// TIA Portal project "Metrou_2026" (V15.1)

(* hardware
DEVICE "S71500/ET200MP station_1"  S7-1500 station
   slot 0: "Rail_0"  Rack  6ES7 590-1***0-0AA0
   slot 1: "PLC_1(Scari)"  CPU 1513-1 PN  6ES7 513-1AL02-0AB0  V2.6
      slot 3: "CPU display_1"  6ES7591-1AA00-0AA0
DEVICE "S71500/ET200MP station_2"  S7-1500 station
   slot 0: "Rail_0"  Rack  6ES7 590-1***0-0AA0
   slot 1: "PLC_1(Metrou)"  CPU 1513-1 PN  6ES7 513-1AL02-0AB0  V2.6
      slot 3: "CPU display_1"  6ES7591-1AA00-0AA0
DEVICE "HMI_1(Scari)"  KTP900 Basic PN
   slot 0: "HMI_1(Scari)"  KTP900 Basic PN  6AV2 123-2JB03-0AX0  15.1.0.0
   slot 1: "HMI_RT_1"  KTP900 Basic PN  6AV2 123-2JB03-0AX0  15.1.0.0
   slot 5: "HMI_1(Scari).IE_CP_1"  PROFINET Interface  15.0.1.0
      slot 1: "PROFINET Interface_1"  PROFINET Interface
         slot 1: "Port_1"  Port
DEVICE "HMI_1(Metrou)"  KTP900 Basic PN
   slot 0: "HMI_1(Metrou)"  KTP900 Basic PN  6AV2 123-2JB03-0AX0  15.1.0.0
   slot 1: "HMI_RT_2"  KTP900 Basic PN  6AV2 123-2JB03-0AX0  15.1.0.0
   slot 5: "HMI_1(Metrou).IE_CP_1"  PROFINET Interface  15.0.1.0
      slot 1: "PROFINET Interface_1"  PROFINET Interface
         slot 1: "Port_1"  Port
*)

// ===== PLC "PLC_1(Scari)"  CPU 1513-1 PN =====

// folder: Alarme/Avarii

DATA_BLOCK "Alarme"   // DB1
{ S7_Optimized_Access := 'TRUE' }
VERSION : 0.1
   VAR
      gather : Word;
      "array" : Array[0..15] of Bool;
   END_VAR
BEGIN
END_DATA_BLOCK

DATA_BLOCK "Avarii"   // DB2
{ S7_Optimized_Access := 'TRUE' }
VERSION : 0.1
   VAR
      esd : Bool;
      btn_esd : Bool;
      reset_esd : Bool;
      avarie_1 : Bool;
      avarie_2 : Bool;
      avarie_3 : Bool;
      avarie_4 : Bool;
      btn_avarie_1 : Bool;
      btn_avarie_2 : Bool;
      btn_avarie_3 : Bool;
      btn_avarie_4 : Bool;
      reset_avarie_1 : Bool;
      reset_avarie_2 : Bool;
      reset_avarie_3 : Bool;
      reset_avarie_4 : Bool;
   END_VAR
BEGIN
END_DATA_BLOCK

// folder: HMI

DATA_BLOCK "HMI"   // DB10
{ S7_Optimized_Access := 'TRUE' }
VERSION : 0.1
   VAR
      motor_stea_1 : Bool;
      motor_triunghi_1 : Bool;
      mod_motor_1 : DInt;   // 0 -> stea, 1 -> triunghi
      pornit_HMI_1 : Bool;
      time_elapsed_HMI_1 : Bool;
      timp_secunde_c_1 : Time;
      timp_secunde_u_1 : Time;
      motor_stea_2 : Bool;
      motor_triunghi_2 : Bool;
      mod_motor_2 : DInt;   // 0 -> stea, 1 -> triunghi
      pornit_HMI_2 : Bool;
      time_elapsed_HMI_2 : Bool;
      timp_secunde_c_2 : Time;
      timp_secunde_u_2 : Time;
      motor_stea_3 : Bool;
      motor_triunghi_3 : Bool;
      mod_motor_3 : DInt;   // 0 -> stea, 1 -> triunghi
      pornit_HMI_3 : Bool;
      time_elapsed_HMI_3 : Bool;
      timp_secunde_c_3 : Time;
      timp_secunde_u_3 : Time;
      motor_stea_4 : Bool;
      motor_triunghi_4 : Bool;
      mod_motor_4 : DInt;   // 0 -> stea, 1 -> triunghi
      pornit_HMI_4 : Bool;
      time_elapsed_HMI_4 : Bool;
      timp_secunde_c_4 : Time;
      timp_secunde_u_4 : Time;
   END_VAR
BEGIN
END_DATA_BLOCK

// folder: Instante

DATA_BLOCK "ESD_Instanta"   // DB4
{ S7_Optimized_Access := 'TRUE' }
VERSION : 0.1
// stored: InstanceOfName Avarei/ESD_FB
"Avarei/ESD_FB"
BEGIN
END_DATA_BLOCK

DATA_BLOCK "Scara1_Instanta_Alarme"   // DB5
{ S7_Optimized_Access := 'TRUE' }
VERSION : 0.1
// stored: InstanceOfName Avarei/ESD_FB
"Avarei/ESD_FB"
BEGIN
END_DATA_BLOCK

DATA_BLOCK "Scara2_Instanta_Alarme"   // DB6
{ S7_Optimized_Access := 'TRUE' }
VERSION : 0.1
// stored: InstanceOfName Avarei/ESD_FB
"Avarei/ESD_FB"
BEGIN
END_DATA_BLOCK

DATA_BLOCK "Scara3_Instanta_Alarme"   // DB7
{ S7_Optimized_Access := 'TRUE' }
VERSION : 0.1
// stored: InstanceOfName Avarei/ESD_FB
"Avarei/ESD_FB"
BEGIN
END_DATA_BLOCK

DATA_BLOCK "Scara4_Instanta_Alarme"   // DB8
{ S7_Optimized_Access := 'TRUE' }
VERSION : 0.1
// stored: InstanceOfName Avarei/ESD_FB
"Avarei/ESD_FB"
BEGIN
END_DATA_BLOCK

DATA_BLOCK "Scara1_Instanta_FB"   // DB9
{ S7_Optimized_Access := 'TRUE' }
VERSION : 0.1
// stored: InstanceOfName Scari
"Scari"
BEGIN
END_DATA_BLOCK

DATA_BLOCK "HMI_Scara_Instanta"   // DB11
{ S7_Optimized_Access := 'TRUE' }
VERSION : 0.1
// stored: InstanceOfName HMI_Scara
"HMI_Scara"
BEGIN
END_DATA_BLOCK

DATA_BLOCK "Scara2_Instanta_FB"   // DB15
{ S7_Optimized_Access := 'TRUE' }
VERSION : 0.1
// stored: InstanceOfName Scari
"Scari"
BEGIN
END_DATA_BLOCK

DATA_BLOCK "Scara4_Instanta_FB"   // DB16
{ S7_Optimized_Access := 'TRUE' }
VERSION : 0.1
// stored: InstanceOfName Scari
"Scari"
BEGIN
END_DATA_BLOCK

DATA_BLOCK "Scara3_Instanta_FB"   // DB17
{ S7_Optimized_Access := 'TRUE' }
VERSION : 0.1
// stored: InstanceOfName Scari
"Scari"
BEGIN
END_DATA_BLOCK

DATA_BLOCK "HMI_Scara2_Instanta"   // DB18
{ S7_Optimized_Access := 'TRUE' }
VERSION : 0.1
// stored: InstanceOfName HMI_Scara
"HMI_Scara"
BEGIN
END_DATA_BLOCK

DATA_BLOCK "HMI_Scara3_Instanta"   // DB19
{ S7_Optimized_Access := 'TRUE' }
VERSION : 0.1
// stored: InstanceOfName HMI_Scara
"HMI_Scara"
BEGIN
END_DATA_BLOCK

DATA_BLOCK "HMI_Scara4_Instanta"   // DB20
{ S7_Optimized_Access := 'TRUE' }
VERSION : 0.1
// stored: InstanceOfName HMI_Scara
"HMI_Scara"
BEGIN
END_DATA_BLOCK

// folder: Scari

DATA_BLOCK "Scara1_DB"   // DB3
{ S7_Optimized_Access := 'TRUE' }
VERSION : 0.1
   VAR
      "mod" : DInt;
      btn_start : Bool;
      btn_stop : Bool;
      senzor_persoana_urcare : Bool;
      senzor_persoana_coborare : Bool;
      stea_urcare : Bool;
      stea_coborare : Bool;
      triunghi_urcare : Bool;
      triunghi_coborare : Bool;
      urcare_HMI : Bool;
      coborare_HMI : Bool;
      et_stea_u : Time;
      et_stea_c : Time;
      et_persoana_u : Time;
      et_persoana_c : Time;
   END_VAR
BEGIN
END_DATA_BLOCK

DATA_BLOCK "Scara2_DB"   // DB12
{ S7_Optimized_Access := 'TRUE' }
VERSION : 0.1
   VAR
      "mod" : DInt;
      btn_start : Bool;
      btn_stop : Bool;
      senzor_persoana_urcare : Bool;
      senzor_persoana_coborare : Bool;
      stea_urcare : Bool;
      stea_coborare : Bool;
      triunghi_urcare : Bool;
      triunghi_coborare : Bool;
      urcare_HMI : Bool;
      coborare_HMI : Bool;
      et_stea_u : Time;
      et_stea_c : Time;
      et_persoana_u : Time;
      et_persoana_c : Time;
   END_VAR
BEGIN
END_DATA_BLOCK

DATA_BLOCK "Scara3_DB"   // DB13
{ S7_Optimized_Access := 'TRUE' }
VERSION : 0.1
   VAR
      "mod" : DInt;
      btn_start : Bool;
      btn_stop : Bool;
      senzor_persoana_urcare : Bool;
      senzor_persoana_coborare : Bool;
      stea_urcare : Bool;
      stea_coborare : Bool;
      triunghi_urcare : Bool;
      triunghi_coborare : Bool;
      urcare_HMI : Bool;
      coborare_HMI : Bool;
      et_stea_u : Time;
      et_stea_c : Time;
      et_persoana_u : Time;
      et_persoana_c : Time;
   END_VAR
BEGIN
END_DATA_BLOCK

DATA_BLOCK "Scara4_DB"   // DB14
{ S7_Optimized_Access := 'TRUE' }
VERSION : 0.1
   VAR
      "mod" : DInt;
      btn_start : Bool;
      btn_stop : Bool;
      senzor_persoana_urcare : Bool;
      senzor_persoana_coborare : Bool;
      stea_urcare : Bool;
      stea_coborare : Bool;
      triunghi_urcare : Bool;
      triunghi_coborare : Bool;
      urcare_HMI : Bool;
      coborare_HMI : Bool;
      et_stea_u : Time;
      et_stea_c : Time;
      et_persoana_u : Time;
      et_persoana_c : Time;
   END_VAR
BEGIN
END_DATA_BLOCK

// folder: (top level)

ORGANIZATION_BLOCK "Main"   // OB1, LAD, ProgramCycle
TITLE = "Main Program Sweep (Cycle)"
{ S7_Optimized_Access := 'TRUE' }
VERSION : 0.1
   VAR_INPUT
      Initial_Call : Bool;   // Initial call of this OB
      Remanence : Bool;   // =True, if remanent data are available
   END_VAR
BEGIN

REGION Network 1: gather de alarme
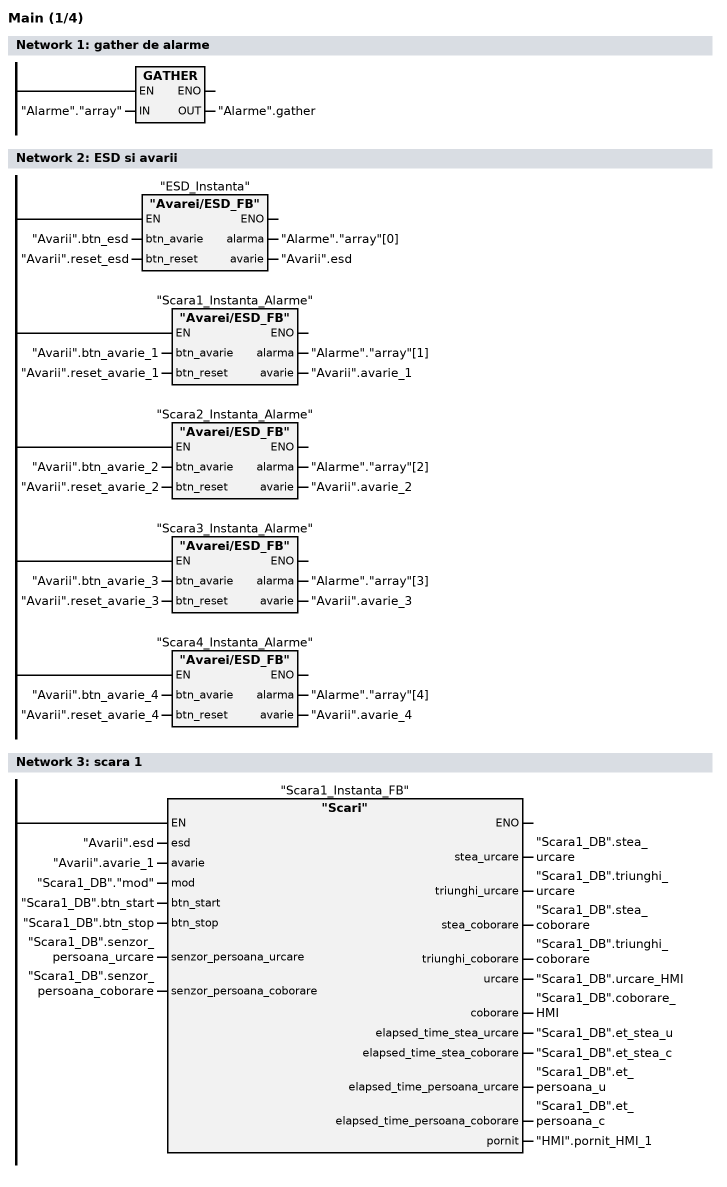
   GATHER(IN := "Alarme"."array", OUT => "Alarme".gather);
END_REGION

REGION Network 2: ESD si avarii
   RUNG wire#powerrail
      "ESD_Instanta"(btn_avarie := "Avarii".btn_esd, btn_reset := "Avarii".reset_esd, alarma => "Alarme"."array"[0], avarie => "Avarii".esd)
   END_RUNG
   RUNG wire#powerrail
      "Scara1_Instanta_Alarme"(btn_avarie := "Avarii".btn_avarie_1, btn_reset := "Avarii".reset_avarie_1, alarma => "Alarme"."array"[1], avarie => "Avarii".avarie_1)
   END_RUNG
   RUNG wire#powerrail
      "Scara2_Instanta_Alarme"(btn_avarie := "Avarii".btn_avarie_2, btn_reset := "Avarii".reset_avarie_2, alarma => "Alarme"."array"[2], avarie => "Avarii".avarie_2)
   END_RUNG
   RUNG wire#powerrail
      "Scara3_Instanta_Alarme"(btn_avarie := "Avarii".btn_avarie_3, btn_reset := "Avarii".reset_avarie_3, alarma => "Alarme"."array"[3], avarie => "Avarii".avarie_3)
   END_RUNG
   RUNG wire#powerrail
      "Scara4_Instanta_Alarme"(btn_avarie := "Avarii".btn_avarie_4, btn_reset := "Avarii".reset_avarie_4, alarma => "Alarme"."array"[4], avarie => "Avarii".avarie_4)
   END_RUNG
   // the same network as SCL:
   "ESD_Instanta"(btn_avarie := "Avarii".btn_esd,   // "Avarei/ESD_FB"
                  btn_reset := "Avarii".reset_esd,
                  alarma => "Alarme"."array"[0],
                  avarie => "Avarii".esd);
   "Scara1_Instanta_Alarme"(btn_avarie := "Avarii".btn_avarie_1,   // "Avarei/ESD_FB"
                           btn_reset := "Avarii".reset_avarie_1,
                           alarma => "Alarme"."array"[1],
                           avarie => "Avarii".avarie_1);
   "Scara2_Instanta_Alarme"(btn_avarie := "Avarii".btn_avarie_2,   // "Avarei/ESD_FB"
                           btn_reset := "Avarii".reset_avarie_2,
                           alarma => "Alarme"."array"[2],
                           avarie => "Avarii".avarie_2);
   "Scara3_Instanta_Alarme"(btn_avarie := "Avarii".btn_avarie_3,   // "Avarei/ESD_FB"
                           btn_reset := "Avarii".reset_avarie_3,
                           alarma => "Alarme"."array"[3],
                           avarie => "Avarii".avarie_3);
   "Scara4_Instanta_Alarme"(btn_avarie := "Avarii".btn_avarie_4,   // "Avarei/ESD_FB"
                           btn_reset := "Avarii".reset_avarie_4,
                           alarma => "Alarme"."array"[4],
                           avarie => "Avarii".avarie_4);
END_REGION

REGION Network 3: scara 1
   RUNG wire#powerrail
      "Scara1_Instanta_FB"(esd := "Avarii".esd, avarie := "Avarii".avarie_1, "mod" := "Scara1_DB"."mod", btn_start := "Scara1_DB".btn_start, btn_stop := "Scara1_DB".btn_stop, senzor_persoana_urcare := "Scara1_DB".senzor_persoana_urcare, senzor_persoana_coborare := "Scara1_DB".senzor_persoana_coborare, stea_urcare => "Scara1_DB".stea_urcare, triunghi_urcare => "Scara1_DB".triunghi_urcare, stea_coborare => "Scara1_DB".stea_coborare, triunghi_coborare => "Scara1_DB".triunghi_coborare, urcare => "Scara1_DB".urcare_HMI, coborare => "Scara1_DB".coborare_HMI, elapsed_time_stea_urcare => "Scara1_DB".et_stea_u, elapsed_time_stea_coborare => "Scara1_DB".et_stea_c, elapsed_time_persoana_urcare => "Scara1_DB".et_persoana_u, elapsed_time_persoana_coborare => "Scara1_DB".et_persoana_c, pornit => "HMI".pornit_HMI_1)
   END_RUNG
   // the same network as SCL:
   "Scara1_Instanta_FB"(esd := "Avarii".esd,   // "Scari"
                        avarie := "Avarii".avarie_1,
                        "mod" := "Scara1_DB"."mod",
                        btn_start := "Scara1_DB".btn_start,
                        btn_stop := "Scara1_DB".btn_stop,
                        senzor_persoana_urcare := "Scara1_DB".senzor_persoana_urcare,
                        senzor_persoana_coborare := "Scara1_DB".senzor_persoana_coborare,
                        stea_urcare => "Scara1_DB".stea_urcare,
                        triunghi_urcare => "Scara1_DB".triunghi_urcare,
                        stea_coborare => "Scara1_DB".stea_coborare,
                        triunghi_coborare => "Scara1_DB".triunghi_coborare,
                        urcare => "Scara1_DB".urcare_HMI,
                        coborare => "Scara1_DB".coborare_HMI,
                        elapsed_time_stea_urcare => "Scara1_DB".et_stea_u,
                        elapsed_time_stea_coborare => "Scara1_DB".et_stea_c,
                        elapsed_time_persoana_urcare => "Scara1_DB".et_persoana_u,
                        elapsed_time_persoana_coborare => "Scara1_DB".et_persoana_c,
                        pornit => "HMI".pornit_HMI_1);
END_REGION

REGION Network 4: HMI scara 1
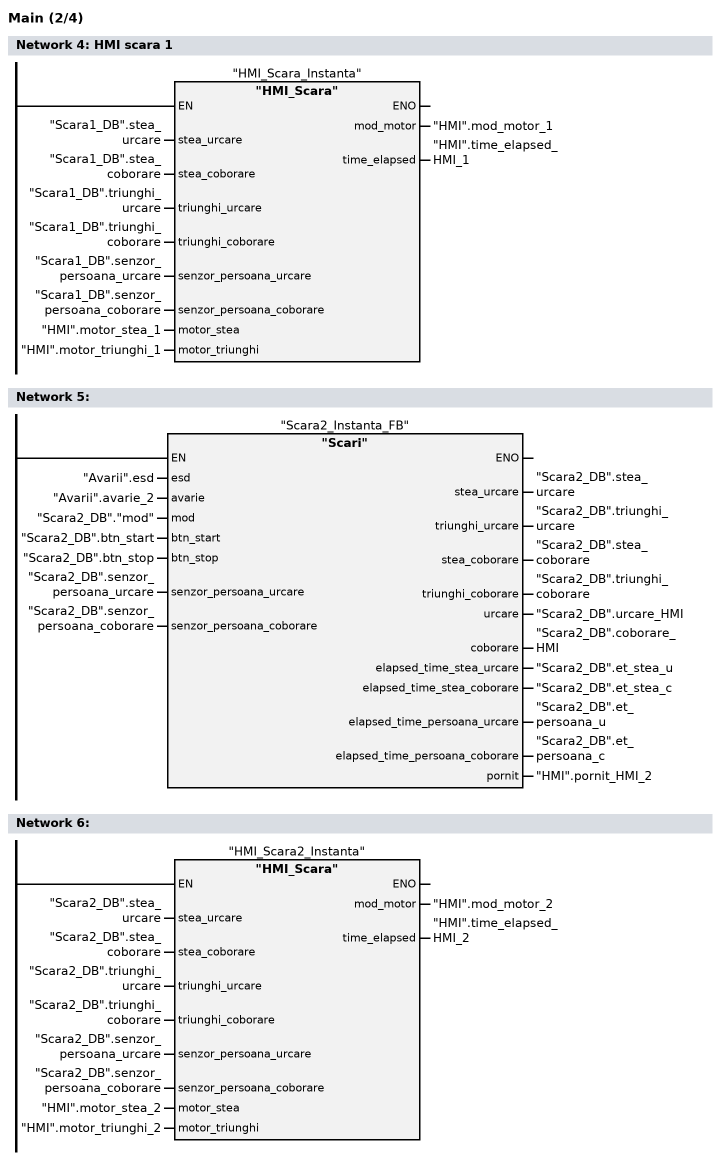
   RUNG wire#powerrail
      "HMI_Scara_Instanta"(stea_urcare := "Scara1_DB".stea_urcare, stea_coborare := "Scara1_DB".stea_coborare, triunghi_urcare := "Scara1_DB".triunghi_urcare, triunghi_coborare := "Scara1_DB".triunghi_coborare, senzor_persoana_urcare := "Scara1_DB".senzor_persoana_urcare, senzor_persoana_coborare := "Scara1_DB".senzor_persoana_coborare, motor_stea := "HMI".motor_stea_1, motor_triunghi := "HMI".motor_triunghi_1, mod_motor => "HMI".mod_motor_1, time_elapsed => "HMI".time_elapsed_HMI_1)
   END_RUNG
   // the same network as SCL:
   "HMI_Scara_Instanta"(stea_urcare := "Scara1_DB".stea_urcare,   // "HMI_Scara"
                        stea_coborare := "Scara1_DB".stea_coborare,
                        triunghi_urcare := "Scara1_DB".triunghi_urcare,
                        triunghi_coborare := "Scara1_DB".triunghi_coborare,
                        senzor_persoana_urcare := "Scara1_DB".senzor_persoana_urcare,
                        senzor_persoana_coborare := "Scara1_DB".senzor_persoana_coborare,
                        motor_stea := "HMI".motor_stea_1,
                        motor_triunghi := "HMI".motor_triunghi_1,
                        mod_motor => "HMI".mod_motor_1,
                        time_elapsed => "HMI".time_elapsed_HMI_1);
END_REGION

REGION Network 5
   RUNG wire#powerrail
      "Scara2_Instanta_FB"(esd := "Avarii".esd, avarie := "Avarii".avarie_2, "mod" := "Scara2_DB"."mod", btn_start := "Scara2_DB".btn_start, btn_stop := "Scara2_DB".btn_stop, senzor_persoana_urcare := "Scara2_DB".senzor_persoana_urcare, senzor_persoana_coborare := "Scara2_DB".senzor_persoana_coborare, stea_urcare => "Scara2_DB".stea_urcare, triunghi_urcare => "Scara2_DB".triunghi_urcare, stea_coborare => "Scara2_DB".stea_coborare, triunghi_coborare => "Scara2_DB".triunghi_coborare, urcare => "Scara2_DB".urcare_HMI, coborare => "Scara2_DB".coborare_HMI, elapsed_time_stea_urcare => "Scara2_DB".et_stea_u, elapsed_time_stea_coborare => "Scara2_DB".et_stea_c, elapsed_time_persoana_urcare => "Scara2_DB".et_persoana_u, elapsed_time_persoana_coborare => "Scara2_DB".et_persoana_c, pornit => "HMI".pornit_HMI_2)
   END_RUNG
   // the same network as SCL:
   "Scara2_Instanta_FB"(esd := "Avarii".esd,   // "Scari"
                        avarie := "Avarii".avarie_2,
                        "mod" := "Scara2_DB"."mod",
                        btn_start := "Scara2_DB".btn_start,
                        btn_stop := "Scara2_DB".btn_stop,
                        senzor_persoana_urcare := "Scara2_DB".senzor_persoana_urcare,
                        senzor_persoana_coborare := "Scara2_DB".senzor_persoana_coborare,
                        stea_urcare => "Scara2_DB".stea_urcare,
                        triunghi_urcare => "Scara2_DB".triunghi_urcare,
                        stea_coborare => "Scara2_DB".stea_coborare,
                        triunghi_coborare => "Scara2_DB".triunghi_coborare,
                        urcare => "Scara2_DB".urcare_HMI,
                        coborare => "Scara2_DB".coborare_HMI,
                        elapsed_time_stea_urcare => "Scara2_DB".et_stea_u,
                        elapsed_time_stea_coborare => "Scara2_DB".et_stea_c,
                        elapsed_time_persoana_urcare => "Scara2_DB".et_persoana_u,
                        elapsed_time_persoana_coborare => "Scara2_DB".et_persoana_c,
                        pornit => "HMI".pornit_HMI_2);
END_REGION

REGION Network 6
   RUNG wire#powerrail
      "HMI_Scara2_Instanta"(stea_urcare := "Scara2_DB".stea_urcare, stea_coborare := "Scara2_DB".stea_coborare, triunghi_urcare := "Scara2_DB".triunghi_urcare, triunghi_coborare := "Scara2_DB".triunghi_coborare, senzor_persoana_urcare := "Scara2_DB".senzor_persoana_urcare, senzor_persoana_coborare := "Scara2_DB".senzor_persoana_coborare, motor_stea := "HMI".motor_stea_2, motor_triunghi := "HMI".motor_triunghi_2, mod_motor => "HMI".mod_motor_2, time_elapsed => "HMI".time_elapsed_HMI_2)
   END_RUNG
   // the same network as SCL:
   "HMI_Scara2_Instanta"(stea_urcare := "Scara2_DB".stea_urcare,   // "HMI_Scara"
                         stea_coborare := "Scara2_DB".stea_coborare,
                         triunghi_urcare := "Scara2_DB".triunghi_urcare,
                         triunghi_coborare := "Scara2_DB".triunghi_coborare,
                         senzor_persoana_urcare := "Scara2_DB".senzor_persoana_urcare,
                         senzor_persoana_coborare := "Scara2_DB".senzor_persoana_coborare,
                         motor_stea := "HMI".motor_stea_2,
                         motor_triunghi := "HMI".motor_triunghi_2,
                         mod_motor => "HMI".mod_motor_2,
                         time_elapsed => "HMI".time_elapsed_HMI_2);
END_REGION

REGION Network 7
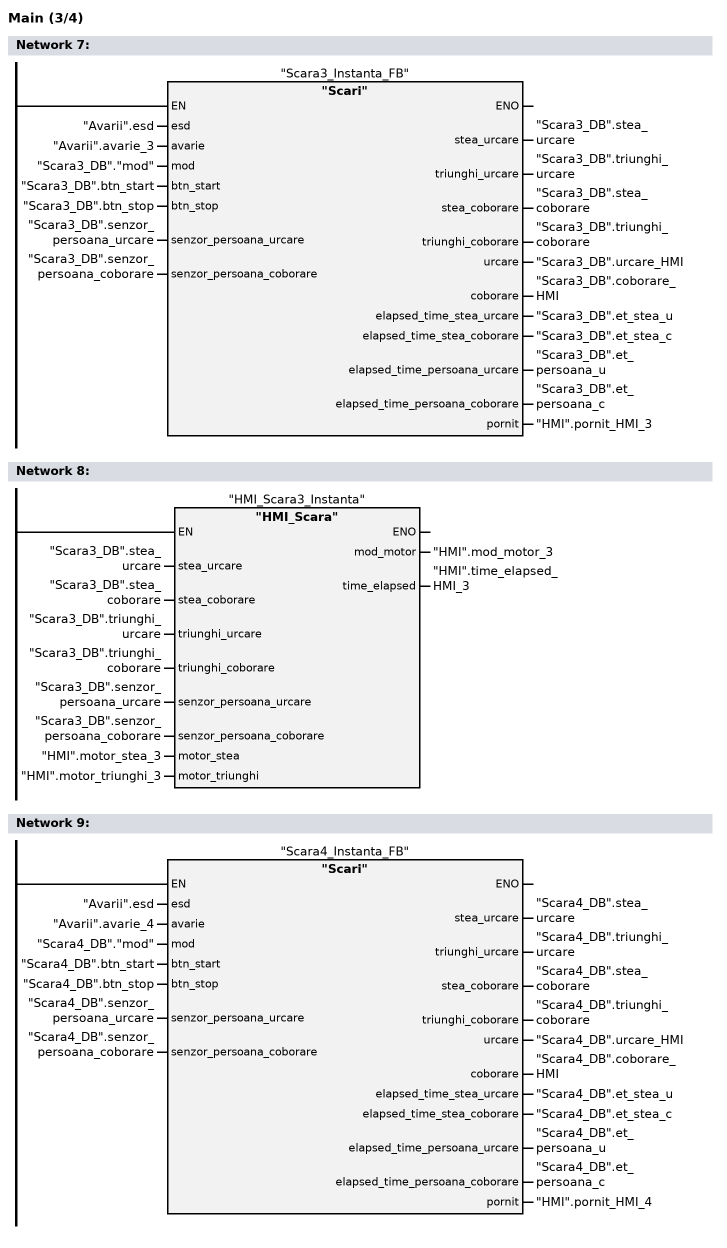
   RUNG wire#powerrail
      "Scara3_Instanta_FB"(esd := "Avarii".esd, avarie := "Avarii".avarie_3, "mod" := "Scara3_DB"."mod", btn_start := "Scara3_DB".btn_start, btn_stop := "Scara3_DB".btn_stop, senzor_persoana_urcare := "Scara3_DB".senzor_persoana_urcare, senzor_persoana_coborare := "Scara3_DB".senzor_persoana_coborare, stea_urcare => "Scara3_DB".stea_urcare, triunghi_urcare => "Scara3_DB".triunghi_urcare, stea_coborare => "Scara3_DB".stea_coborare, triunghi_coborare => "Scara3_DB".triunghi_coborare, urcare => "Scara3_DB".urcare_HMI, coborare => "Scara3_DB".coborare_HMI, elapsed_time_stea_urcare => "Scara3_DB".et_stea_u, elapsed_time_stea_coborare => "Scara3_DB".et_stea_c, elapsed_time_persoana_urcare => "Scara3_DB".et_persoana_u, elapsed_time_persoana_coborare => "Scara3_DB".et_persoana_c, pornit => "HMI".pornit_HMI_3)
   END_RUNG
   // the same network as SCL:
   "Scara3_Instanta_FB"(esd := "Avarii".esd,   // "Scari"
                        avarie := "Avarii".avarie_3,
                        "mod" := "Scara3_DB"."mod",
                        btn_start := "Scara3_DB".btn_start,
                        btn_stop := "Scara3_DB".btn_stop,
                        senzor_persoana_urcare := "Scara3_DB".senzor_persoana_urcare,
                        senzor_persoana_coborare := "Scara3_DB".senzor_persoana_coborare,
                        stea_urcare => "Scara3_DB".stea_urcare,
                        triunghi_urcare => "Scara3_DB".triunghi_urcare,
                        stea_coborare => "Scara3_DB".stea_coborare,
                        triunghi_coborare => "Scara3_DB".triunghi_coborare,
                        urcare => "Scara3_DB".urcare_HMI,
                        coborare => "Scara3_DB".coborare_HMI,
                        elapsed_time_stea_urcare => "Scara3_DB".et_stea_u,
                        elapsed_time_stea_coborare => "Scara3_DB".et_stea_c,
                        elapsed_time_persoana_urcare => "Scara3_DB".et_persoana_u,
                        elapsed_time_persoana_coborare => "Scara3_DB".et_persoana_c,
                        pornit => "HMI".pornit_HMI_3);
END_REGION

REGION Network 8
   RUNG wire#powerrail
      "HMI_Scara3_Instanta"(stea_urcare := "Scara3_DB".stea_urcare, stea_coborare := "Scara3_DB".stea_coborare, triunghi_urcare := "Scara3_DB".triunghi_urcare, triunghi_coborare := "Scara3_DB".triunghi_coborare, senzor_persoana_urcare := "Scara3_DB".senzor_persoana_urcare, senzor_persoana_coborare := "Scara3_DB".senzor_persoana_coborare, motor_stea := "HMI".motor_stea_3, motor_triunghi := "HMI".motor_triunghi_3, mod_motor => "HMI".mod_motor_3, time_elapsed => "HMI".time_elapsed_HMI_3)
   END_RUNG
   // the same network as SCL:
   "HMI_Scara3_Instanta"(stea_urcare := "Scara3_DB".stea_urcare,   // "HMI_Scara"
                         stea_coborare := "Scara3_DB".stea_coborare,
                         triunghi_urcare := "Scara3_DB".triunghi_urcare,
                         triunghi_coborare := "Scara3_DB".triunghi_coborare,
                         senzor_persoana_urcare := "Scara3_DB".senzor_persoana_urcare,
                         senzor_persoana_coborare := "Scara3_DB".senzor_persoana_coborare,
                         motor_stea := "HMI".motor_stea_3,
                         motor_triunghi := "HMI".motor_triunghi_3,
                         mod_motor => "HMI".mod_motor_3,
                         time_elapsed => "HMI".time_elapsed_HMI_3);
END_REGION

REGION Network 9
   RUNG wire#powerrail
      "Scara4_Instanta_FB"(esd := "Avarii".esd, avarie := "Avarii".avarie_4, "mod" := "Scara4_DB"."mod", btn_start := "Scara4_DB".btn_start, btn_stop := "Scara4_DB".btn_stop, senzor_persoana_urcare := "Scara4_DB".senzor_persoana_urcare, senzor_persoana_coborare := "Scara4_DB".senzor_persoana_coborare, stea_urcare => "Scara4_DB".stea_urcare, triunghi_urcare => "Scara4_DB".triunghi_urcare, stea_coborare => "Scara4_DB".stea_coborare, triunghi_coborare => "Scara4_DB".triunghi_coborare, urcare => "Scara4_DB".urcare_HMI, coborare => "Scara4_DB".coborare_HMI, elapsed_time_stea_urcare => "Scara4_DB".et_stea_u, elapsed_time_stea_coborare => "Scara4_DB".et_stea_c, elapsed_time_persoana_urcare => "Scara4_DB".et_persoana_u, elapsed_time_persoana_coborare => "Scara4_DB".et_persoana_c, pornit => "HMI".pornit_HMI_4)
   END_RUNG
   // the same network as SCL:
   "Scara4_Instanta_FB"(esd := "Avarii".esd,   // "Scari"
                        avarie := "Avarii".avarie_4,
                        "mod" := "Scara4_DB"."mod",
                        btn_start := "Scara4_DB".btn_start,
                        btn_stop := "Scara4_DB".btn_stop,
                        senzor_persoana_urcare := "Scara4_DB".senzor_persoana_urcare,
                        senzor_persoana_coborare := "Scara4_DB".senzor_persoana_coborare,
                        stea_urcare => "Scara4_DB".stea_urcare,
                        triunghi_urcare => "Scara4_DB".triunghi_urcare,
                        stea_coborare => "Scara4_DB".stea_coborare,
                        triunghi_coborare => "Scara4_DB".triunghi_coborare,
                        urcare => "Scara4_DB".urcare_HMI,
                        coborare => "Scara4_DB".coborare_HMI,
                        elapsed_time_stea_urcare => "Scara4_DB".et_stea_u,
                        elapsed_time_stea_coborare => "Scara4_DB".et_stea_c,
                        elapsed_time_persoana_urcare => "Scara4_DB".et_persoana_u,
                        elapsed_time_persoana_coborare => "Scara4_DB".et_persoana_c,
                        pornit => "HMI".pornit_HMI_4);
END_REGION

REGION Network 10
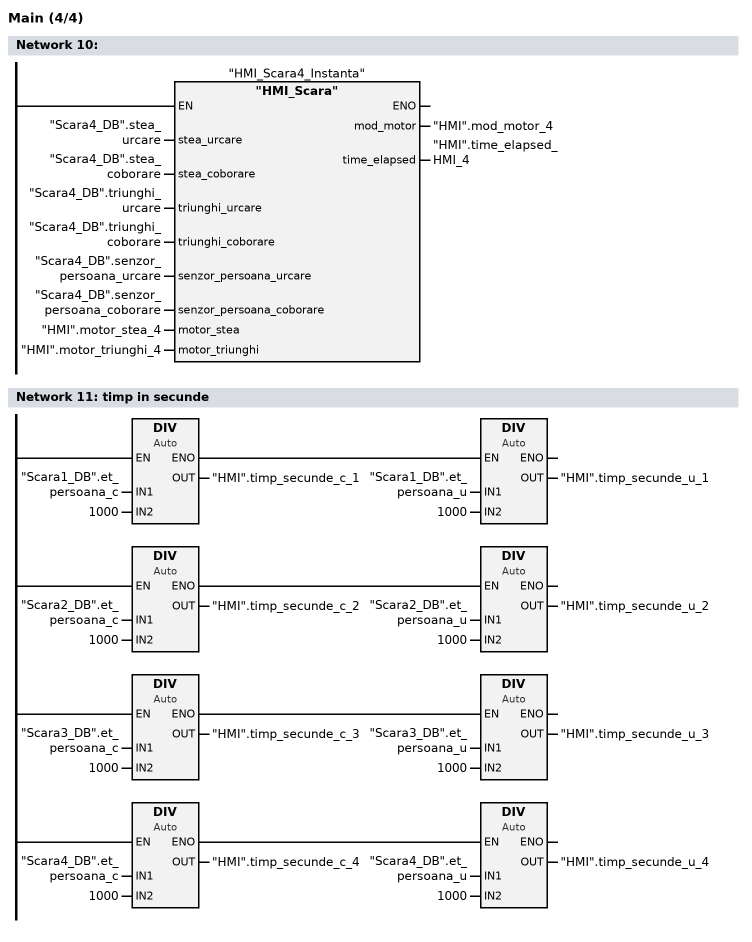
   RUNG wire#powerrail
      "HMI_Scara4_Instanta"(stea_urcare := "Scara4_DB".stea_urcare, stea_coborare := "Scara4_DB".stea_coborare, triunghi_urcare := "Scara4_DB".triunghi_urcare, triunghi_coborare := "Scara4_DB".triunghi_coborare, senzor_persoana_urcare := "Scara4_DB".senzor_persoana_urcare, senzor_persoana_coborare := "Scara4_DB".senzor_persoana_coborare, motor_stea := "HMI".motor_stea_4, motor_triunghi := "HMI".motor_triunghi_4, mod_motor => "HMI".mod_motor_4, time_elapsed => "HMI".time_elapsed_HMI_4)
   END_RUNG
   // the same network as SCL:
   "HMI_Scara4_Instanta"(stea_urcare := "Scara4_DB".stea_urcare,   // "HMI_Scara"
                         stea_coborare := "Scara4_DB".stea_coborare,
                         triunghi_urcare := "Scara4_DB".triunghi_urcare,
                         triunghi_coborare := "Scara4_DB".triunghi_coborare,
                         senzor_persoana_urcare := "Scara4_DB".senzor_persoana_urcare,
                         senzor_persoana_coborare := "Scara4_DB".senzor_persoana_coborare,
                         motor_stea := "HMI".motor_stea_4,
                         motor_triunghi := "HMI".motor_triunghi_4,
                         mod_motor => "HMI".mod_motor_4,
                         time_elapsed => "HMI".time_elapsed_HMI_4);
END_REGION

REGION Network 11: timp in secunde
   RUNG wire#powerrail
      Div(in1 := "Scara1_DB".et_persoana_c, in2 := 1000, out => "HMI".timp_secunde_c_1)
      Div(in1 := "Scara1_DB".et_persoana_u, in2 := 1000, out => "HMI".timp_secunde_u_1)
   END_RUNG
   RUNG wire#powerrail
      Div(in1 := "Scara2_DB".et_persoana_c, in2 := 1000, out => "HMI".timp_secunde_c_2)
      Div(in1 := "Scara2_DB".et_persoana_u, in2 := 1000, out => "HMI".timp_secunde_u_2)
   END_RUNG
   RUNG wire#powerrail
      Div(in1 := "Scara3_DB".et_persoana_c, in2 := 1000, out => "HMI".timp_secunde_c_3)
      Div(in1 := "Scara3_DB".et_persoana_u, in2 := 1000, out => "HMI".timp_secunde_u_3)
   END_RUNG
   RUNG wire#powerrail
      Div(in1 := "Scara4_DB".et_persoana_c, in2 := 1000, out => "HMI".timp_secunde_c_4)
      Div(in1 := "Scara4_DB".et_persoana_u, in2 := 1000, out => "HMI".timp_secunde_u_4)
   END_RUNG
   // the same network as SCL:
   "HMI".timp_secunde_c_1 := "Scara1_DB".et_persoana_c / 1000;
   "HMI".timp_secunde_u_1 := "Scara1_DB".et_persoana_u / 1000;
   "HMI".timp_secunde_c_2 := "Scara2_DB".et_persoana_c / 1000;
   "HMI".timp_secunde_u_2 := "Scara2_DB".et_persoana_u / 1000;
   "HMI".timp_secunde_c_3 := "Scara3_DB".et_persoana_c / 1000;
   "HMI".timp_secunde_u_3 := "Scara3_DB".et_persoana_u / 1000;
   "HMI".timp_secunde_c_4 := "Scara4_DB".et_persoana_c / 1000;
   "HMI".timp_secunde_u_4 := "Scara4_DB".et_persoana_u / 1000;
END_REGION
END_ORGANIZATION_BLOCK

// folder: Alarme/Avarii

FUNCTION_BLOCK "Avarei/ESD_FB"   // FB2, LAD
{ S7_Optimized_Access := 'TRUE' }
VERSION : 0.1
   VAR_OUTPUT
      alarma : Bool;
      avarie : Bool;
   END_VAR
   VAR_IN_OUT
      btn_avarie : Bool;
      btn_reset : Bool;
   END_VAR
   VAR
      ton : TON_TIME;
   END_VAR
BEGIN

REGION Network 1: seteaza avaria
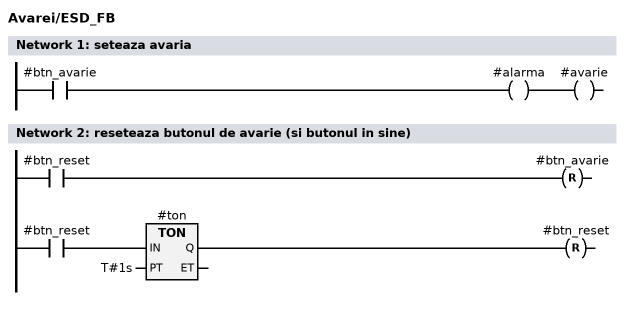
   RUNG wire#powerrail
      Contact( #btn_avarie )
      Coil( #alarma )
      Coil( #avarie )
   END_RUNG
   // the same network as SCL:
   #alarma := #btn_avarie;
   #avarie := #btn_avarie;
END_REGION

REGION Network 2: reseteaza butonul de avarie (si butonul in sine)
   IF #btn_reset THEN #btn_avarie := FALSE; END_IF;
   #ton(IN := #btn_reset, PT := T#1s);   // TON
   IF #ton.Q THEN #btn_reset := FALSE; END_IF;
END_REGION
END_FUNCTION_BLOCK

// folder: HMI

FUNCTION_BLOCK "HMI_Scara"   // FB3, LAD
{ S7_Optimized_Access := 'TRUE' }
VERSION : 0.1
   VAR_INPUT
      stea_urcare : Bool;
      stea_coborare : Bool;
      triunghi_urcare : Bool;
      triunghi_coborare : Bool;
      senzor_persoana_urcare : Bool;
      senzor_persoana_coborare : Bool;
   END_VAR
   VAR_OUTPUT
      mod_motor : DInt;
      time_elapsed : Bool;
   END_VAR
   VAR_IN_OUT
      motor_stea : Bool;
      motor_triunghi : Bool;
   END_VAR
BEGIN

REGION Network 1
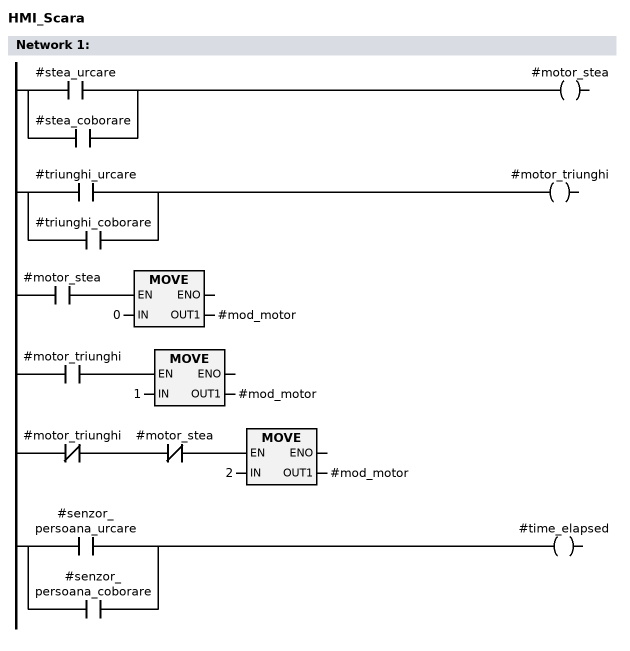
   RUNG wire#powerrail
      Contact( #stea_urcare )
      wire#w1
      Coil( #motor_stea )
   END_RUNG
   RUNG wire#powerrail
      Contact( #stea_coborare )
   END_RUNG wire#w1
   RUNG wire#powerrail
      Contact( #triunghi_urcare )
      wire#w2
      Coil( #motor_triunghi )
   END_RUNG
   RUNG wire#powerrail
      Contact( #triunghi_coborare )
   END_RUNG wire#w2
   RUNG wire#powerrail
      Contact( #motor_stea )
      Move(in := 0, out1 => #mod_motor)
   END_RUNG
   RUNG wire#powerrail
      Contact( #motor_triunghi )
      Move(in := 1, out1 => #mod_motor)
   END_RUNG
   RUNG wire#powerrail
      I_Contact( #motor_triunghi )
      I_Contact( #motor_stea )
      Move(in := 2, out1 => #mod_motor)
   END_RUNG
   RUNG wire#powerrail
      Contact( #senzor_persoana_urcare )
      wire#w3
      Coil( #time_elapsed )
   END_RUNG
   RUNG wire#powerrail
      Contact( #senzor_persoana_coborare )
   END_RUNG wire#w3
   // the same network as SCL:
   #motor_stea := #stea_urcare OR #stea_coborare;
   #motor_triunghi := #triunghi_urcare OR #triunghi_coborare;
   IF #motor_stea THEN #mod_motor := 0; END_IF;
   IF #motor_triunghi THEN #mod_motor := 1; END_IF;
   IF NOT #motor_triunghi AND NOT #motor_stea THEN #mod_motor := 2; END_IF;
   #time_elapsed := #senzor_persoana_urcare OR #senzor_persoana_coborare;
END_REGION
END_FUNCTION_BLOCK

// folder: Scari

FUNCTION_BLOCK "Scari"   // FB1, LAD
{ S7_Optimized_Access := 'TRUE' }
VERSION : 0.1
   VAR_INPUT
      esd : Bool;
      avarie : Bool;
      "mod" : DInt;
   END_VAR
   VAR_OUTPUT
      stea_urcare : Bool;
      triunghi_urcare : Bool;
      stea_coborare : Bool;
      triunghi_coborare : Bool;
      urcare : Bool;
      coborare : Bool;
      elapsed_time_stea_urcare : Time;
      elapsed_time_stea_coborare : Time;
      elapsed_time_persoana_urcare : Time;
      elapsed_time_persoana_coborare : Time;
      pornit : Bool;
   END_VAR
   VAR_IN_OUT
      btn_start : Bool;
      btn_stop : Bool;
      senzor_persoana_urcare : Bool;
      senzor_persoana_coborare : Bool;
   END_VAR
   VAR
      ton_stea_urcare : TON_TIME;
      ton_stea_coborare : TON_TIME;
      ton_persoana_urcare : TON_TIME;
      ton_persoana_coborare : TON_TIME;
      ton_btn_stop : TON_TIME;
      permisiune_urcare : Bool;
      permisiune_coborare : Bool;
      plecare_stea_urcare : Bool;
      plecare_stea_coborare : Bool;
      plecare_triunghi_urcare : Bool;
      plecare_triunghi_coborare : Bool;
      terminat_timer_stea_urcare : Bool;
      terminat_timer_stea_coborare : Bool;
      terminat_persoana_urcare : Bool;
      terminat_persoana_coborare : Bool;
      trecut_regim_stea_u : Bool;
      trecut_regim_stea_c : Bool;
   END_VAR
BEGIN

REGION Network 1: Reseteaza senzorii daca modul nu este setat
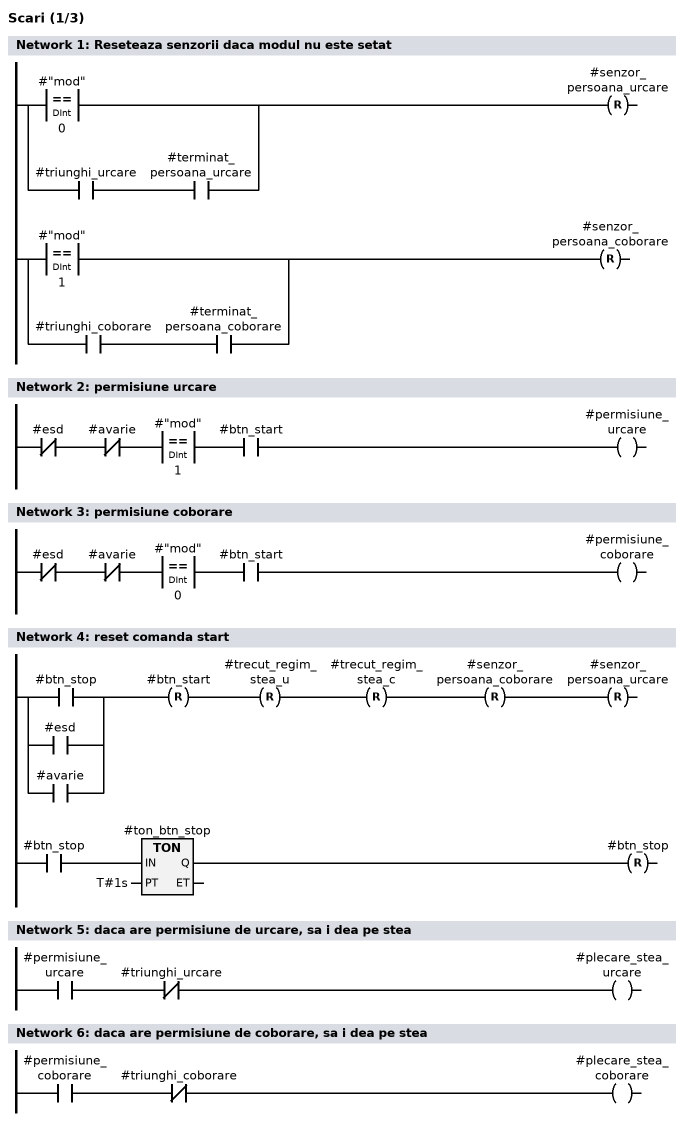
   RUNG wire#powerrail
      { S7_Templates := "SrcType := DInt" } EQ_Contact(in1 := #"mod", in2 := 0)
      wire#w1
      R_Coil( #senzor_persoana_urcare )
   END_RUNG
   RUNG wire#powerrail
      Contact( #triunghi_urcare )
      Contact( #terminat_persoana_urcare )
   END_RUNG wire#w1
   RUNG wire#powerrail
      { S7_Templates := "SrcType := DInt" } EQ_Contact(in1 := #"mod", in2 := 1)
      wire#w2
      R_Coil( #senzor_persoana_coborare )
   END_RUNG
   RUNG wire#powerrail
      Contact( #triunghi_coborare )
      Contact( #terminat_persoana_coborare )
   END_RUNG wire#w2
   // the same network as SCL:
   IF (#"mod" = 0) OR (#triunghi_urcare AND #terminat_persoana_urcare) THEN
       #senzor_persoana_urcare := FALSE;
   END_IF;
   IF (#"mod" = 1) OR (#triunghi_coborare AND #terminat_persoana_coborare) THEN
       #senzor_persoana_coborare := FALSE;
   END_IF;
END_REGION

REGION Network 2: permisiune urcare
   RUNG wire#powerrail
      I_Contact( #esd )
      I_Contact( #avarie )
      { S7_Templates := "SrcType := DInt" } EQ_Contact(in1 := #"mod", in2 := 1)
      Contact( #btn_start )
      Coil( #permisiune_urcare )
   END_RUNG
   // the same network as SCL:
   #permisiune_urcare := NOT #esd AND NOT #avarie AND (#"mod" = 1) AND #btn_start;
END_REGION

REGION Network 3: permisiune coborare
   RUNG wire#powerrail
      I_Contact( #esd )
      I_Contact( #avarie )
      { S7_Templates := "SrcType := DInt" } EQ_Contact(in1 := #"mod", in2 := 0)
      Contact( #btn_start )
      Coil( #permisiune_coborare )
   END_RUNG
   // the same network as SCL:
   #permisiune_coborare := NOT #esd AND NOT #avarie AND (#"mod" = 0) AND #btn_start;
END_REGION

REGION Network 4: reset comanda start
   IF #btn_stop OR #esd OR #avarie THEN
       #btn_start := FALSE;
       #trecut_regim_stea_u := FALSE;
       #trecut_regim_stea_c := FALSE;
       #senzor_persoana_coborare := FALSE;
       #senzor_persoana_urcare := FALSE;
   END_IF;
   #ton_btn_stop(IN := #btn_stop, PT := T#1s);   // TON
   IF #ton_btn_stop.Q THEN #btn_stop := FALSE; END_IF;
END_REGION

REGION Network 5: daca are permisiune de urcare, sa i dea pe stea
   RUNG wire#powerrail
      Contact( #permisiune_urcare )
      I_Contact( #triunghi_urcare )
      Coil( #plecare_stea_urcare )
   END_RUNG
   // the same network as SCL:
   #plecare_stea_urcare := #permisiune_urcare AND NOT #triunghi_urcare;
END_REGION

REGION Network 6: daca are permisiune de coborare, sa i dea pe stea
   RUNG wire#powerrail
      Contact( #permisiune_coborare )
      I_Contact( #triunghi_coborare )
      Coil( #plecare_stea_coborare )
   END_RUNG
   // the same network as SCL:
   #plecare_stea_coborare := #permisiune_coborare AND NOT #triunghi_coborare;
END_REGION

REGION Network 7: daca e pe stea/triunghi, sa dea si pe output
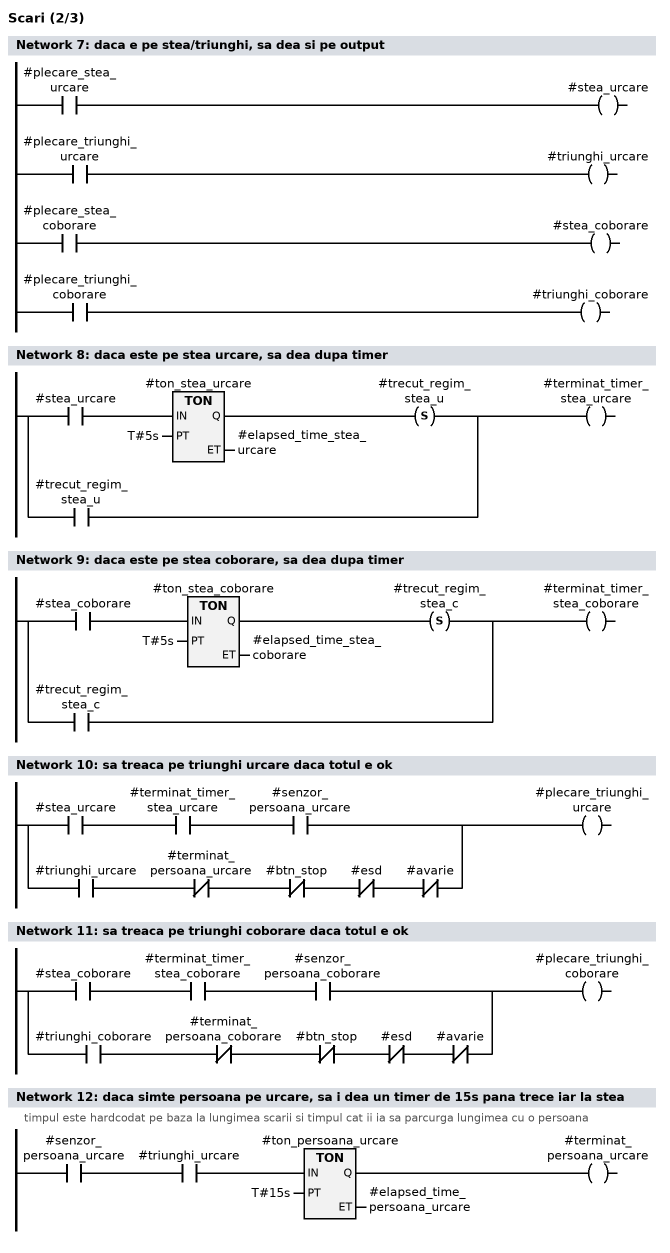
   RUNG wire#powerrail
      Contact( #plecare_stea_urcare )
      Coil( #stea_urcare )
   END_RUNG
   RUNG wire#powerrail
      Contact( #plecare_triunghi_urcare )
      Coil( #triunghi_urcare )
   END_RUNG
   RUNG wire#powerrail
      Contact( #plecare_stea_coborare )
      Coil( #stea_coborare )
   END_RUNG
   RUNG wire#powerrail
      Contact( #plecare_triunghi_coborare )
      Coil( #triunghi_coborare )
   END_RUNG
   // the same network as SCL:
   #stea_urcare := #plecare_stea_urcare;
   #triunghi_urcare := #plecare_triunghi_urcare;
   #stea_coborare := #plecare_stea_coborare;
   #triunghi_coborare := #plecare_triunghi_coborare;
END_REGION

REGION Network 8: daca este pe stea urcare, sa dea dupa timer
   #ton_stea_urcare(IN := #stea_urcare, PT := T#5s, ET => #elapsed_time_stea_urcare);   // TON
   IF #ton_stea_urcare.Q THEN #trecut_regim_stea_u := TRUE; END_IF;
   #terminat_timer_stea_urcare := #ton_stea_urcare.Q OR #trecut_regim_stea_u;
END_REGION

REGION Network 9: daca este pe stea coborare, sa dea dupa timer
   #ton_stea_coborare(IN := #stea_coborare, PT := T#5s, ET => #elapsed_time_stea_coborare);   // TON
   IF #ton_stea_coborare.Q THEN #trecut_regim_stea_c := TRUE; END_IF;
   #terminat_timer_stea_coborare := #ton_stea_coborare.Q OR #trecut_regim_stea_c;
END_REGION

REGION Network 10: sa treaca pe triunghi urcare daca totul e ok
   RUNG wire#powerrail
      Contact( #stea_urcare )
      Contact( #terminat_timer_stea_urcare )
      Contact( #senzor_persoana_urcare )
      wire#w1
      Coil( #plecare_triunghi_urcare )
   END_RUNG
   RUNG wire#powerrail
      Contact( #triunghi_urcare )
      I_Contact( #terminat_persoana_urcare )
      I_Contact( #btn_stop )
      I_Contact( #esd )
      I_Contact( #avarie )
   END_RUNG wire#w1
   // the same network as SCL:
   #plecare_triunghi_urcare := (#stea_urcare AND #terminat_timer_stea_urcare AND #senzor_persoana_urcare) OR (#triunghi_urcare AND NOT #terminat_persoana_urcare AND NOT #btn_stop AND NOT #esd AND NOT #avarie);
END_REGION

REGION Network 11: sa treaca pe triunghi coborare daca totul e ok
   RUNG wire#powerrail
      Contact( #stea_coborare )
      Contact( #terminat_timer_stea_coborare )
      Contact( #senzor_persoana_coborare )
      wire#w1
      Coil( #plecare_triunghi_coborare )
   END_RUNG
   RUNG wire#powerrail
      Contact( #triunghi_coborare )
      I_Contact( #terminat_persoana_coborare )
      I_Contact( #btn_stop )
      I_Contact( #esd )
      I_Contact( #avarie )
   END_RUNG wire#w1
   // the same network as SCL:
   #plecare_triunghi_coborare := (#stea_coborare AND #terminat_timer_stea_coborare AND #senzor_persoana_coborare) OR (#triunghi_coborare AND NOT #terminat_persoana_coborare AND NOT #btn_stop AND NOT #esd AND NOT #avarie);
END_REGION

REGION Network 12: daca simte persoana pe urcare, sa i dea un timer de 15s pana trece iar la stea
   // timpul este hardcodat pe baza la lungimea scarii si timpul cat ii ia sa parcurga lungimea cu o persoana
   #ton_persoana_urcare(IN := #senzor_persoana_urcare AND #triunghi_urcare,   // TON
                        PT := T#15s,
                        ET => #elapsed_time_persoana_urcare);
   #terminat_persoana_urcare := #ton_persoana_urcare.Q;
END_REGION

REGION Network 13: daca simte persoana pe coborare, sa i dea un timer de 15s pana trece iar la stea
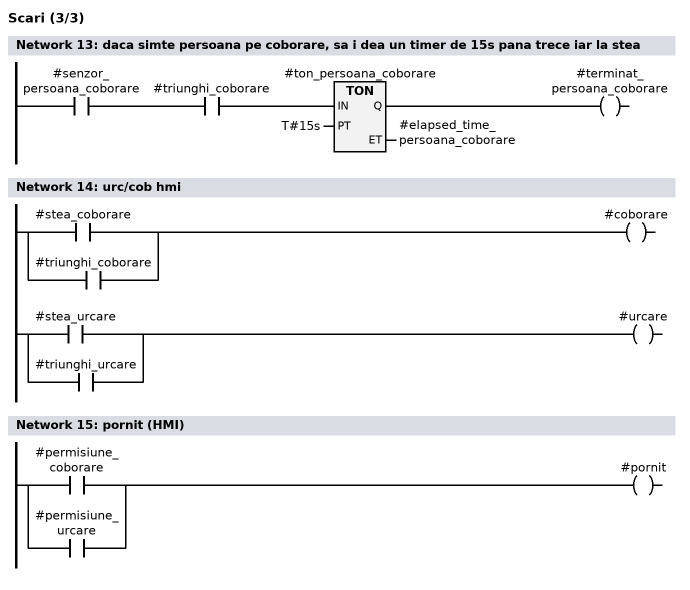
   #ton_persoana_coborare(IN := #senzor_persoana_coborare AND #triunghi_coborare,   // TON
                          PT := T#15s,
                          ET => #elapsed_time_persoana_coborare);
   #terminat_persoana_coborare := #ton_persoana_coborare.Q;
END_REGION

REGION Network 14: urc/cob hmi
   RUNG wire#powerrail
      Contact( #stea_coborare )
      wire#w1
      Coil( #coborare )
   END_RUNG
   RUNG wire#powerrail
      Contact( #triunghi_coborare )
   END_RUNG wire#w1
   RUNG wire#powerrail
      Contact( #stea_urcare )
      wire#w2
      Coil( #urcare )
   END_RUNG
   RUNG wire#powerrail
      Contact( #triunghi_urcare )
   END_RUNG wire#w2
   // the same network as SCL:
   #coborare := #stea_coborare OR #triunghi_coborare;
   #urcare := #stea_urcare OR #triunghi_urcare;
END_REGION

REGION Network 15: pornit (HMI)
   RUNG wire#powerrail
      Contact( #permisiune_coborare )
      wire#w1
      Coil( #pornit )
   END_RUNG
   RUNG wire#powerrail
      Contact( #permisiune_urcare )
   END_RUNG wire#w1
   // the same network as SCL:
   #pornit := #permisiune_coborare OR #permisiune_urcare;
END_REGION
END_FUNCTION_BLOCK

// ===== PLC "PLC_1(Metrou)"  CPU 1513-1 PN =====

VAR_GLOBAL   // PLC tag table "Default tag table"
   "Clock_Byte" AT %MB8080 : Byte;
   "Clock_10Hz" AT %M8080.0 : Bool;
   "Clock_5Hz" AT %M8080.1 : Bool;
   "Clock_2.5Hz" AT %M8080.2 : Bool;
   "Clock_2Hz" AT %M8080.3 : Bool;
   "Clock_1.25Hz" AT %M8080.4 : Bool;
   "Clock_1Hz" AT %M8080.5 : Bool;
   "Clock_0.625Hz" AT %M8080.6 : Bool;
   "Clock_0.5Hz" AT %M8080.7 : Bool;
END_VAR

// folder: Avarii/Alarme

DATA_BLOCK "Avarii"   // DB1
{ S7_Optimized_Access := 'TRUE' }
VERSION : 0.1
   VAR
      esd : Bool;
      btn_esd : Bool;
      reset_esd : Bool;
      avarie_usa_1 : Bool;
      btn_avarie_usa_1 : Bool;
      reset_avaie_usa_1 : Bool;
      avarie_usa_2 : Bool;
      btn_avarie_usa_2 : Bool;
      reset_avaie_usa_2 : Bool;
      avarie_usa_3 : Bool;
      btn_avarie_usa_3 : Bool;
      reset_avaie_usa_3 : Bool;
   END_VAR
BEGIN
END_DATA_BLOCK

DATA_BLOCK "Alarme"   // DB2
{ S7_Optimized_Access := 'TRUE' }
VERSION : 0.1
   VAR
      gather : Word;
      "array" : Array[0..15] of Bool;
   END_VAR
BEGIN
END_DATA_BLOCK

// folder: Instante

DATA_BLOCK "Usa_Metrou_DB_1"   // DB4
{ S7_Optimized_Access := 'TRUE' }
VERSION : 0.1
// stored: InstanceOfName Usa_Metrou
"Usa_Metrou"
BEGIN
END_DATA_BLOCK

DATA_BLOCK "Alarma_Avarie_FB_DB_ESD"   // DB5
{ S7_Optimized_Access := 'TRUE' }
VERSION : 0.1
// stored: InstanceOfName Alarma_Avarie_FB
"Alarma_Avarie_FB"
BEGIN
END_DATA_BLOCK

DATA_BLOCK "Alarma_Avarie_FB_DB_Usa1"   // DB6
{ S7_Optimized_Access := 'TRUE' }
VERSION : 0.1
// stored: InstanceOfName Alarma_Avarie_FB
"Alarma_Avarie_FB"
BEGIN
END_DATA_BLOCK

DATA_BLOCK "Alarma_Avarie_FB_Usa2"   // DB7
{ S7_Optimized_Access := 'TRUE' }
VERSION : 0.1
// stored: InstanceOfName Alarma_Avarie_FB
"Alarma_Avarie_FB"
BEGIN
END_DATA_BLOCK

DATA_BLOCK "Alarma_Avarie_FB_DB_Usa3"   // DB8
{ S7_Optimized_Access := 'TRUE' }
VERSION : 0.1
// stored: InstanceOfName Alarma_Avarie_FB
"Alarma_Avarie_FB"
BEGIN
END_DATA_BLOCK

// folder: Usa_Metrou

DATA_BLOCK "Usa_Metrou1_DB"   // DB3
{ S7_Optimized_Access := 'TRUE' }
VERSION : 0.1
   VAR
      "mod" : DInt;
      vizibilitate_mod_02 : Bool;
      confirmare_primita : Bool;
      trimite_confirmare : Bool;
      senzor_laser_1 : Bool;
      senzor_laser_2 : Bool;
      deschide_1 : Bool;
      deschide_2 : Bool;
      usi_inchise : Bool;
      sunet_buzzer : Bool;
      secventa_intrare : Bool;
      secventa_iesire : Bool;
      secventa_pornita : Bool;
   END_VAR
BEGIN
END_DATA_BLOCK

// folder: (top level)

ORGANIZATION_BLOCK "Main"   // OB1, LAD, ProgramCycle
TITLE = "Main Program Sweep (Cycle)"
{ S7_Optimized_Access := 'TRUE' }
VERSION : 0.1
   VAR_INPUT
      Initial_Call : Bool;   // Initial call of this OB
      Remanence : Bool;   // =True, if remanent data are available
   END_VAR
BEGIN

REGION Network 1: gather pt alarme
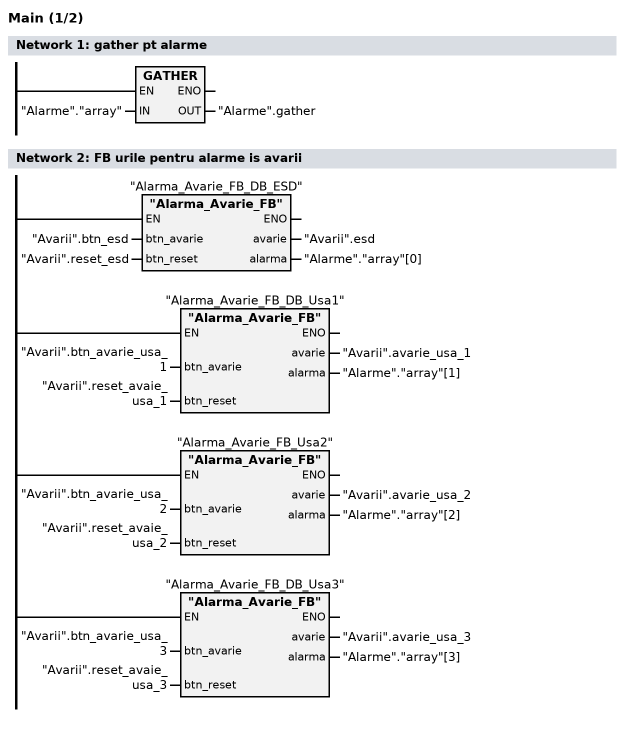
   GATHER(IN := "Alarme"."array", OUT => "Alarme".gather);
END_REGION

REGION Network 2: FB urile pentru alarme is avarii
   RUNG wire#powerrail
      "Alarma_Avarie_FB_DB_ESD"(btn_avarie := "Avarii".btn_esd, btn_reset := "Avarii".reset_esd, avarie => "Avarii".esd, alarma => "Alarme"."array"[0])
   END_RUNG
   RUNG wire#powerrail
      "Alarma_Avarie_FB_DB_Usa1"(btn_avarie := "Avarii".btn_avarie_usa_1, btn_reset := "Avarii".reset_avaie_usa_1, avarie => "Avarii".avarie_usa_1, alarma => "Alarme"."array"[1])
   END_RUNG
   RUNG wire#powerrail
      "Alarma_Avarie_FB_Usa2"(btn_avarie := "Avarii".btn_avarie_usa_2, btn_reset := "Avarii".reset_avaie_usa_2, avarie => "Avarii".avarie_usa_2, alarma => "Alarme"."array"[2])
   END_RUNG
   RUNG wire#powerrail
      "Alarma_Avarie_FB_DB_Usa3"(btn_avarie := "Avarii".btn_avarie_usa_3, btn_reset := "Avarii".reset_avaie_usa_3, avarie => "Avarii".avarie_usa_3, alarma => "Alarme"."array"[3])
   END_RUNG
   // the same network as SCL:
   "Alarma_Avarie_FB_DB_ESD"(btn_avarie := "Avarii".btn_esd,   // "Alarma_Avarie_FB"
                           btn_reset := "Avarii".reset_esd,
                           avarie => "Avarii".esd,
                           alarma => "Alarme"."array"[0]);
   "Alarma_Avarie_FB_DB_Usa1"(btn_avarie := "Avarii".btn_avarie_usa_1,   // "Alarma_Avarie_FB"
                           btn_reset := "Avarii".reset_avaie_usa_1,
                           avarie => "Avarii".avarie_usa_1,
                           alarma => "Alarme"."array"[1]);
   "Alarma_Avarie_FB_Usa2"(btn_avarie := "Avarii".btn_avarie_usa_2,   // "Alarma_Avarie_FB"
                           btn_reset := "Avarii".reset_avaie_usa_2,
                           avarie => "Avarii".avarie_usa_2,
                           alarma => "Alarme"."array"[2]);
   "Alarma_Avarie_FB_DB_Usa3"(btn_avarie := "Avarii".btn_avarie_usa_3,   // "Alarma_Avarie_FB"
                           btn_reset := "Avarii".reset_avaie_usa_3,
                           avarie => "Avarii".avarie_usa_3,
                           alarma => "Alarme"."array"[3]);
END_REGION

REGION Network 3: usa 1 metrou
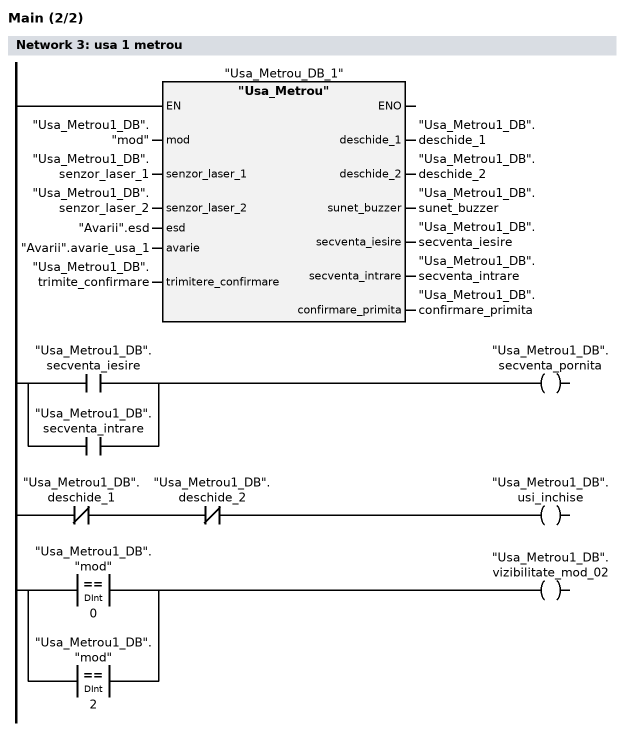
   RUNG wire#powerrail
      "Usa_Metrou_DB_1"("mod" := "Usa_Metrou1_DB"."mod", senzor_laser_1 := "Usa_Metrou1_DB".senzor_laser_1, senzor_laser_2 := "Usa_Metrou1_DB".senzor_laser_2, esd := "Avarii".esd, avarie := "Avarii".avarie_usa_1, trimitere_confirmare := "Usa_Metrou1_DB".trimite_confirmare, deschide_1 => "Usa_Metrou1_DB".deschide_1, deschide_2 => "Usa_Metrou1_DB".deschide_2, sunet_buzzer => "Usa_Metrou1_DB".sunet_buzzer, secventa_iesire => "Usa_Metrou1_DB".secventa_iesire, secventa_intrare => "Usa_Metrou1_DB".secventa_intrare, confirmare_primita => "Usa_Metrou1_DB".confirmare_primita)
   END_RUNG
   RUNG wire#powerrail
      Contact( "Usa_Metrou1_DB".secventa_iesire )
      wire#w1
      Coil( "Usa_Metrou1_DB".secventa_pornita )
   END_RUNG
   RUNG wire#powerrail
      Contact( "Usa_Metrou1_DB".secventa_intrare )
   END_RUNG wire#w1
   RUNG wire#powerrail
      I_Contact( "Usa_Metrou1_DB".deschide_1 )
      I_Contact( "Usa_Metrou1_DB".deschide_2 )
      Coil( "Usa_Metrou1_DB".usi_inchise )
   END_RUNG
   RUNG wire#powerrail
      { S7_Templates := "SrcType := DInt" } EQ_Contact(in1 := "Usa_Metrou1_DB"."mod", in2 := 0)
      wire#w2
      Coil( "Usa_Metrou1_DB".vizibilitate_mod_02 )
   END_RUNG
   RUNG wire#powerrail
      { S7_Templates := "SrcType := DInt" } EQ_Contact(in1 := "Usa_Metrou1_DB"."mod", in2 := 2)
   END_RUNG wire#w2
   // the same network as SCL:
   "Usa_Metrou_DB_1"("mod" := "Usa_Metrou1_DB"."mod",   // "Usa_Metrou"
                     senzor_laser_1 := "Usa_Metrou1_DB".senzor_laser_1,
                     senzor_laser_2 := "Usa_Metrou1_DB".senzor_laser_2,
                     esd := "Avarii".esd,
                     avarie := "Avarii".avarie_usa_1,
                     trimitere_confirmare := "Usa_Metrou1_DB".trimite_confirmare,
                     deschide_1 => "Usa_Metrou1_DB".deschide_1,
                     deschide_2 => "Usa_Metrou1_DB".deschide_2,
                     sunet_buzzer => "Usa_Metrou1_DB".sunet_buzzer,
                     secventa_iesire => "Usa_Metrou1_DB".secventa_iesire,
                     secventa_intrare => "Usa_Metrou1_DB".secventa_intrare,
                     confirmare_primita => "Usa_Metrou1_DB".confirmare_primita);
   "Usa_Metrou1_DB".secventa_pornita := "Usa_Metrou1_DB".secventa_iesire OR "Usa_Metrou1_DB".secventa_intrare;
   "Usa_Metrou1_DB".usi_inchise := NOT "Usa_Metrou1_DB".deschide_1 AND NOT "Usa_Metrou1_DB".deschide_2;
   "Usa_Metrou1_DB".vizibilitate_mod_02 := ("Usa_Metrou1_DB"."mod" = 0) OR ("Usa_Metrou1_DB"."mod" = 2);
END_REGION
END_ORGANIZATION_BLOCK

// folder: Avarii/Alarme

FUNCTION_BLOCK "Alarma_Avarie_FB"   // FB3, LAD
{ S7_Optimized_Access := 'TRUE' }
VERSION : 0.1
   VAR_OUTPUT
      avarie : Bool;
      alarma : Bool;
   END_VAR
   VAR_IN_OUT
      btn_avarie : Bool;
      btn_reset : Bool;
   END_VAR
BEGIN

REGION Network 1: seteaza alarma
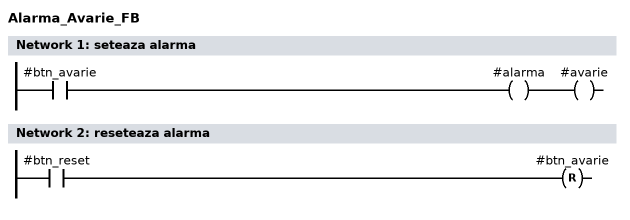
   RUNG wire#powerrail
      Contact( #btn_avarie )
      Coil( #alarma )
      Coil( #avarie )
   END_RUNG
   // the same network as SCL:
   #alarma := #btn_avarie;
   #avarie := #btn_avarie;
END_REGION

REGION Network 2: reseteaza alarma
   RUNG wire#powerrail
      Contact( #btn_reset )
      R_Coil( #btn_avarie )
   END_RUNG
   // the same network as SCL:
   IF #btn_reset THEN #btn_avarie := FALSE; END_IF;
END_REGION
END_FUNCTION_BLOCK

// folder: Buzzer

FUNCTION_BLOCK "Buzzer"   // FB2, LAD
{ S7_Optimized_Access := 'TRUE' }
VERSION : 0.1
   VAR_OUTPUT
      sunet : Bool;
   END_VAR
   VAR
      repeta : Bool;
      auxiliar : Bool;
   END_VAR
   VAR_TEMP   // added for the SCL form of the ladder/FBD networks
      _w1 : Bool;
   END_VAR
BEGIN

REGION Network 1: clock pt SR latch
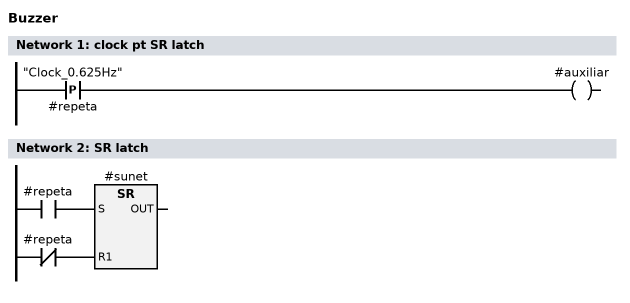
   RUNG wire#powerrail
      P_Contact(operand := "Clock_0.625Hz", bit := #repeta)
      Coil( #auxiliar )
   END_RUNG
   // the same network as SCL:
   #_w1 := "Clock_0.625Hz" AND NOT #repeta;   // rising edge of "Clock_0.625Hz"
   #repeta := "Clock_0.625Hz";
   #auxiliar := #_w1;
END_REGION

REGION Network 2: SR latch
   RUNG wire#powerrail
      Contact( #repeta )
      S_SR(operand := #sunet, r1 := wire#w1)
   END_RUNG
   RUNG wire#powerrail
      I_Contact( #repeta )
   END_RUNG wire#w1
   // the same network as SCL:
   IF #repeta THEN
       #sunet := TRUE;   // SR flip-flop
   END_IF;
   IF NOT #repeta THEN #sunet := FALSE; END_IF;
END_REGION
END_FUNCTION_BLOCK

// folder: Usa_Metrou

FUNCTION_BLOCK "Usa_Metrou"   // FB1, LAD
{ S7_Optimized_Access := 'TRUE' }
VERSION : 0.1
   VAR_INPUT
      "mod" : DInt;
      senzor_laser_1 : Bool;
      senzor_laser_2 : Bool;
      esd : Bool;
      avarie : Bool;
   END_VAR
   VAR_OUTPUT
      deschide_1 : Bool;
      deschide_2 : Bool;
      sunet_buzzer : Bool;
      secventa_iesire : Bool;
      secventa_intrare : Bool;
      confirmare_primita : Bool;
   END_VAR
   VAR_IN_OUT
      trimitere_confirmare : Bool;
   END_VAR
   VAR
      timer_confirmare : TON_TIME;
      timer_deschis_iesire : TON_TIME;
      timer_deschis_intrare : TON_TIME;
      timer_deschis_ambele_parti : TON_TIME;
      Buzzer_Instance : "Buzzer";
      porneste_buzzer : Bool;
      aux1 : Bool;
      aux2 : Bool;
      re1 : Bool;
      re2 : Bool;
      "counter" : DInt;
   END_VAR
   VAR_TEMP   // added for the SCL form of the ladder/FBD networks
      _w1 : Bool;
      _w2 : Bool;
   END_VAR
BEGIN

REGION Network 1: daca are permisiunea, porneste buzzerul
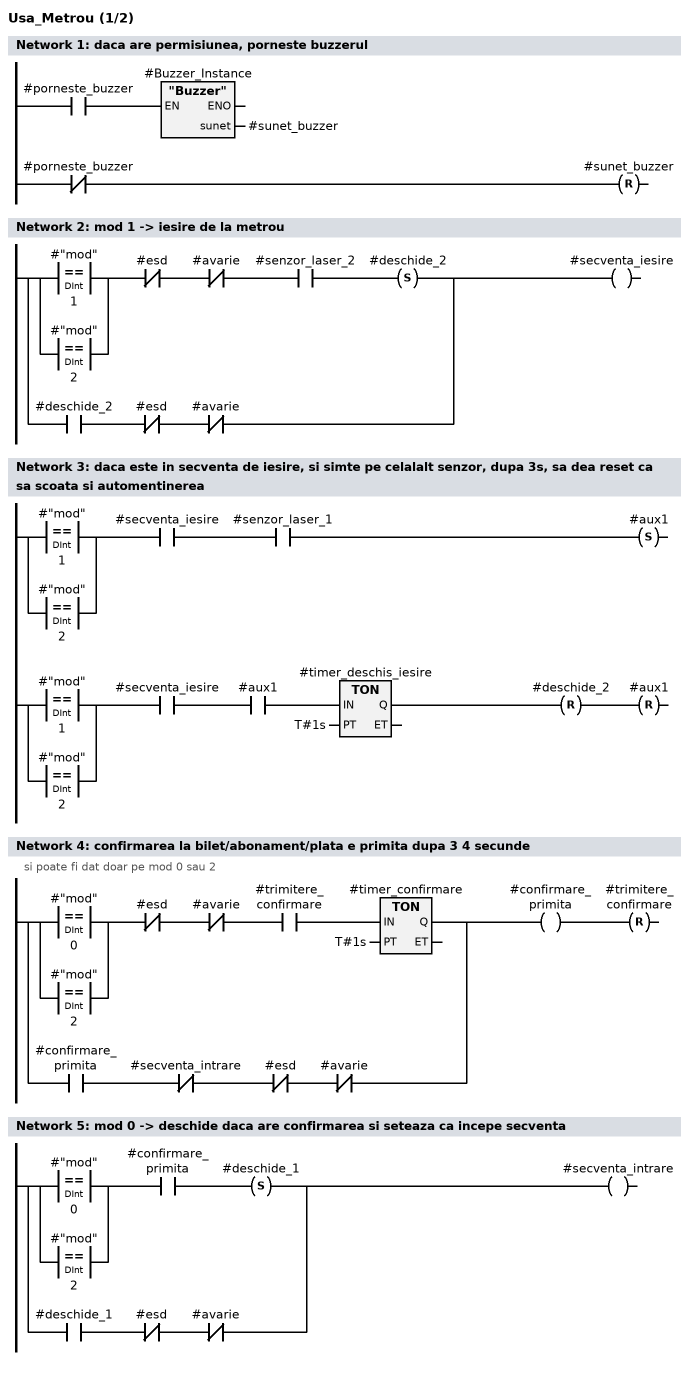
   RUNG wire#powerrail
      Contact( #porneste_buzzer )
      #Buzzer_Instance(sunet => #sunet_buzzer)
   END_RUNG
   RUNG wire#powerrail
      I_Contact( #porneste_buzzer )
      R_Coil( #sunet_buzzer )
   END_RUNG
   // the same network as SCL:
   IF #porneste_buzzer THEN
       #Buzzer_Instance(sunet => #sunet_buzzer);   // "Buzzer"
   END_IF;
   IF NOT #porneste_buzzer THEN #sunet_buzzer := FALSE; END_IF;
END_REGION

REGION Network 2: mod 1 -> iesire de la metrou
   RUNG wire#powerrail
      { S7_Templates := "SrcType := DInt" } EQ_Contact(in1 := #"mod", in2 := 1)
      wire#w1
      I_Contact( #esd )
      I_Contact( #avarie )
      Contact( #senzor_laser_2 )
      S_Coil( #deschide_2 )
      wire#w2
      Coil( #secventa_iesire )
   END_RUNG
   RUNG wire#powerrail
      { S7_Templates := "SrcType := DInt" } EQ_Contact(in1 := #"mod", in2 := 2)
   END_RUNG wire#w1
   RUNG wire#powerrail
      Contact( #deschide_2 )
      I_Contact( #esd )
      I_Contact( #avarie )
   END_RUNG wire#w2
   // the same network as SCL:
   #_w1 := ((#"mod" = 1) OR (#"mod" = 2)) AND NOT #esd AND NOT #avarie AND #senzor_laser_2;
   IF #_w1 THEN #deschide_2 := TRUE; END_IF;
   #secventa_iesire := #_w1 OR (#deschide_2 AND NOT #esd AND NOT #avarie);
END_REGION

REGION Network 3: daca este in secventa de iesire, si simte pe celalalt senzor, dupa 3s, sa dea reset ca sa scoata si automentinerea
   IF ((#"mod" = 1) OR (#"mod" = 2)) AND #secventa_iesire AND #senzor_laser_1 THEN #aux1 := TRUE; END_IF;
   #timer_deschis_iesire(IN := ((#"mod" = 1) OR (#"mod" = 2)) AND #secventa_iesire AND #aux1, PT := T#1s);   // TON
   IF #timer_deschis_iesire.Q THEN
       #deschide_2 := FALSE;
       #aux1 := FALSE;
   END_IF;
END_REGION

REGION Network 4: confirmarea la bilet/abonament/plata e primita dupa 3 4 secunde
   // si poate fi dat doar pe mod 0 sau 2
   #timer_confirmare(IN := ((#"mod" = 0) OR (#"mod" = 2)) AND NOT #esd AND NOT #avarie AND #trimitere_confirmare,   // TON
                     PT := T#1s);
   #confirmare_primita := #timer_confirmare.Q OR (#confirmare_primita AND NOT #secventa_intrare AND NOT #esd AND NOT #avarie);
   IF #confirmare_primita THEN #trimitere_confirmare := FALSE; END_IF;
END_REGION

REGION Network 5: mod 0 -> deschide daca are confirmarea si seteaza ca incepe secventa
   RUNG wire#powerrail
      { S7_Templates := "SrcType := DInt" } EQ_Contact(in1 := #"mod", in2 := 0)
      wire#w1
      Contact( #confirmare_primita )
      S_Coil( #deschide_1 )
      wire#w2
      Coil( #secventa_intrare )
   END_RUNG
   RUNG wire#powerrail
      { S7_Templates := "SrcType := DInt" } EQ_Contact(in1 := #"mod", in2 := 2)
   END_RUNG wire#w1
   RUNG wire#powerrail
      Contact( #deschide_1 )
      I_Contact( #esd )
      I_Contact( #avarie )
   END_RUNG wire#w2
   // the same network as SCL:
   #_w1 := ((#"mod" = 0) OR (#"mod" = 2)) AND #confirmare_primita;
   IF #_w1 THEN #deschide_1 := TRUE; END_IF;
   #secventa_intrare := #_w1 OR (#deschide_1 AND NOT #esd AND NOT #avarie);
END_REGION

REGION Network 6: increment is daca e cazul, da pe buzzer
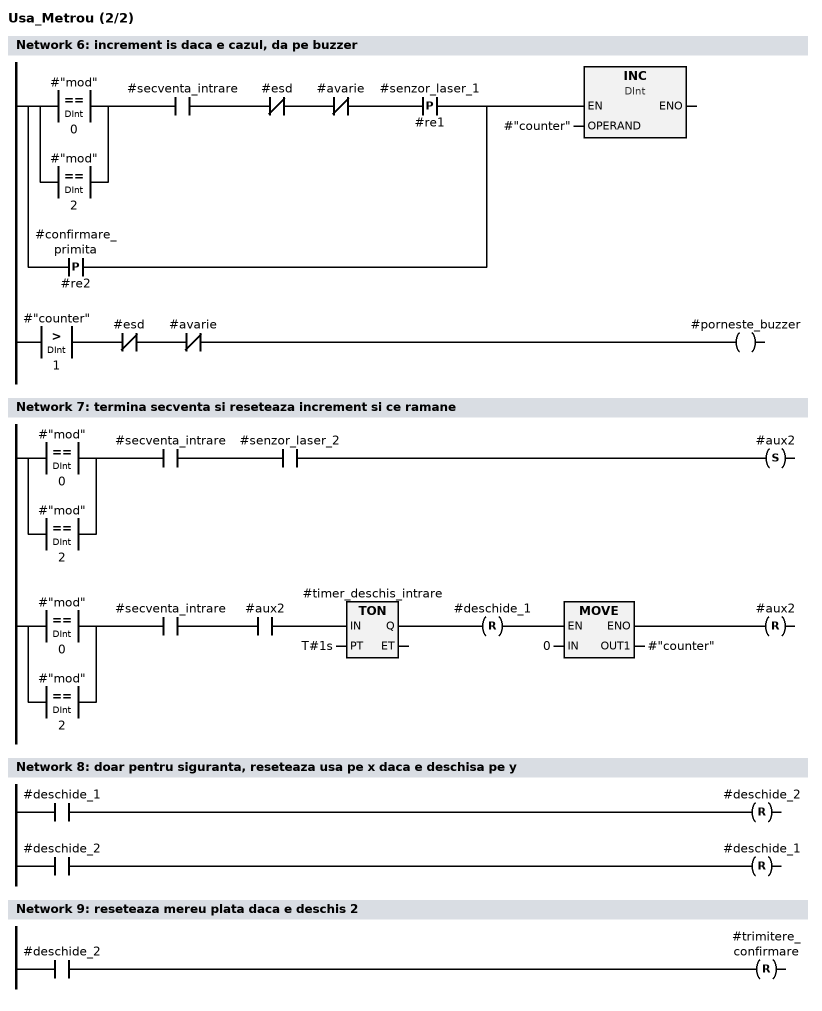
   RUNG wire#powerrail
      { S7_Templates := "SrcType := DInt" } EQ_Contact(in1 := #"mod", in2 := 0)
      wire#w1
      Contact( #secventa_intrare )
      I_Contact( #esd )
      I_Contact( #avarie )
      P_Contact(operand := #senzor_laser_1, bit := #re1)
      wire#w2
      { S7_Templates := "DestType := DInt" } Inc( #"counter" )
   END_RUNG
   RUNG wire#powerrail
      { S7_Templates := "SrcType := DInt" } EQ_Contact(in1 := #"mod", in2 := 2)
   END_RUNG wire#w1
   RUNG wire#powerrail
      P_Contact(operand := #confirmare_primita, bit := #re2)
   END_RUNG wire#w2
   RUNG wire#powerrail
      { S7_Templates := "SrcType := DInt" } GT_Contact(in1 := #"counter", in2 := 1)
      I_Contact( #esd )
      I_Contact( #avarie )
      Coil( #porneste_buzzer )
   END_RUNG
   // the same network as SCL:
   #_w1 := ((#"mod" = 0) OR (#"mod" = 2)) AND #secventa_intrare AND NOT #esd AND NOT #avarie AND #senzor_laser_1 AND NOT #re1;   // rising edge of #senzor_laser_1
   #re1 := #senzor_laser_1;
   #_w2 := #confirmare_primita AND NOT #re2;   // rising edge of #confirmare_primita
   #re2 := #confirmare_primita;
   IF #_w1 OR #_w2 THEN #"counter" := #"counter" + 1; END_IF;
   #porneste_buzzer := (#"counter" > 1) AND NOT #esd AND NOT #avarie;
END_REGION

REGION Network 7: termina secventa si reseteaza increment si ce ramane
   IF ((#"mod" = 0) OR (#"mod" = 2)) AND #secventa_intrare AND #senzor_laser_2 THEN #aux2 := TRUE; END_IF;
   #timer_deschis_intrare(IN := ((#"mod" = 0) OR (#"mod" = 2)) AND #secventa_intrare AND #aux2, PT := T#1s);   // TON
   IF #timer_deschis_intrare.Q THEN
       #deschide_1 := FALSE;
       #"counter" := 0;
       #aux2 := FALSE;
   END_IF;
END_REGION

REGION Network 8: doar pentru siguranta, reseteaza usa pe x daca e deschisa pe y
   RUNG wire#powerrail
      Contact( #deschide_1 )
      R_Coil( #deschide_2 )
   END_RUNG
   RUNG wire#powerrail
      Contact( #deschide_2 )
      R_Coil( #deschide_1 )
   END_RUNG
   // the same network as SCL:
   IF #deschide_1 THEN #deschide_2 := FALSE; END_IF;
   IF #deschide_2 THEN #deschide_1 := FALSE; END_IF;
END_REGION

REGION Network 9: reseteaza mereu plata daca e deschis 2
   RUNG wire#powerrail
      Contact( #deschide_2 )
      R_Coil( #trimitere_confirmare )
   END_RUNG
   // the same network as SCL:
   IF #deschide_2 THEN #trimitere_confirmare := FALSE; END_IF;
END_REGION
END_FUNCTION_BLOCK

(* ===== HMI "HMI_RT_1" =====
system functions are stored by id; their names below are inferred from use
connection "HMI_Connection_1": ETHERNET, SMART_S7_1500_OMS

HMI tags "Default tag table"
   "Alarme_gather" : Word = PLC Alarme.gather, 1 s
   "Avarii_esd" : Bool = PLC Avarii.esd, 1 s
   "Avarii_avarie_1" : Bool = PLC Avarii.avarie_1, 1 s
   "Avarii_btn_esd" : Bool = PLC Avarii.btn_esd, 1 s
   "Avarii_btn_avarie_1" : Bool = PLC Avarii.btn_avarie_1, 1 s
   "Avarii_reset_esd" : Bool = PLC Avarii.reset_esd, 1 s
   "Avarii_reset_avarie_1" : Bool = PLC Avarii.reset_avarie_1, 1 s
   "Scara1_DB_urcare_HMI" : Bool = PLC Scara1_DB.urcare_HMI, 1 s
   "Scara1_DB_coborare_HMI" : Bool = PLC Scara1_DB.coborare_HMI, 1 s
   "HMI_mod_motor" : DInt = PLC HMI.mod_motor_1, 1 s
   "Scara1_DB_mod" : DInt = PLC Scara1_DB.mod, 1 s
   "Scara1_DB_btn_start" : Bool = PLC Scara1_DB.btn_start, 1 s
   "Scara1_DB_btn_stop" : Bool = PLC Scara1_DB.btn_stop, 1 s
   "HMI_pornit_HMI" : Bool = PLC HMI.pornit_HMI_1, 1 s
   "Scara1_DB_senzor_persoana_urcare" : Bool = PLC Scara1_DB.senzor_persoana_urcare, 1 s
   "Scara1_DB_senzor_persoana_coborare" : Bool = PLC Scara1_DB.senzor_persoana_coborare, 1 s
   "HMI_time_elapsed_HMI" : Bool = PLC HMI.time_elapsed_HMI_1, 1 s
   "Scara1_DB_et_persoana_u" : Time = PLC Scara1_DB.et_persoana_u, 1 s
   "Scara1_DB_et_persoana_c" : Time = PLC Scara1_DB.et_persoana_c, 1 s
   "HMI_timp_secunde_c_1" : Time = PLC HMI.timp_secunde_c_1, 1 s
   "HMI_timp_secunde_u_1" : Time = PLC HMI.timp_secunde_u_1, 1 s
   "Avarii_avarie_2" : Bool = PLC Avarii.avarie_2, 1 s
   "Avarii_avarie_3" : Bool = PLC Avarii.avarie_3, 1 s
   "Avarii_avarie_4" : Bool = PLC Avarii.avarie_4, 1 s
   "Avarii_btn_avarie_2" : Bool = PLC Avarii.btn_avarie_2, 1 s
   "Avarii_btn_avarie_3" : Bool = PLC Avarii.btn_avarie_3, 1 s
   "Avarii_btn_avarie_4" : Bool = PLC Avarii.btn_avarie_4, 1 s
   "Avarii_reset_avarie_4" : Bool = PLC Avarii.reset_avarie_4, 1 s
   "Avarii_reset_avarie_3" : Bool = PLC Avarii.reset_avarie_3, 1 s
   "Scara2_DB_urcare_HMI" : Bool = PLC Scara2_DB.urcare_HMI, 1 s
   "Scara2_DB_coborare_HMI" : Bool = PLC Scara2_DB.coborare_HMI, 1 s
   "Scara3_DB_urcare_HMI" : Bool = PLC Scara3_DB.urcare_HMI, 1 s
   "Scara3_DB_coborare_HMI" : Bool = PLC Scara3_DB.coborare_HMI, 1 s
   "Scara4_DB_urcare_HMI" : Bool = PLC Scara4_DB.urcare_HMI, 1 s
   "Scara4_DB_coborare_HMI" : Bool = PLC Scara4_DB.coborare_HMI, 1 s
   "HMI_mod_motor_2" : DInt = PLC HMI.mod_motor_2, 1 s
   "HMI_mod_motor_3" : DInt = PLC HMI.mod_motor_3, 1 s
   "HMI_mod_motor_4" : DInt = PLC HMI.mod_motor_4, 1 s
   "Scara2_DB_mod" : DInt = PLC Scara2_DB.mod, 1 s
   "Scara3_DB_mod" : DInt = PLC Scara3_DB.mod, 1 s
   "Scara4_DB_mod" : DInt = PLC Scara4_DB.mod, 1 s
   "Scara2_DB_btn_start" : Bool = PLC Scara2_DB.btn_start, 1 s
   "Scara3_DB_btn_start" : Bool = PLC Scara3_DB.btn_start, 1 s
   "Scara4_DB_btn_start" : Bool = PLC Scara4_DB.btn_start, 1 s
   "Scara4_DB_btn_stop" : Bool = PLC Scara4_DB.btn_stop, 1 s
   "Scara3_DB_btn_stop" : Bool = PLC Scara3_DB.btn_stop, 1 s
   "Scara2_DB_btn_stop" : Bool = PLC Scara2_DB.btn_stop, 1 s
   "HMI_pornit_HMI_2" : Bool = PLC HMI.pornit_HMI_2, 1 s
   "HMI_pornit_HMI_3" : Bool = PLC HMI.pornit_HMI_3, 1 s
   "HMI_pornit_HMI_4" : Bool = PLC HMI.pornit_HMI_4, 1 s
   "HMI_time_elapsed_HMI_2" : Bool = PLC HMI.time_elapsed_HMI_2, 1 s
   "HMI_time_elapsed_HMI_3" : Bool = PLC HMI.time_elapsed_HMI_3, 1 s
   "HMI_time_elapsed_HMI_4" : Bool = PLC HMI.time_elapsed_HMI_4, 1 s
   "Scara2_DB_senzor_persoana_urcare" : Bool = PLC Scara2_DB.senzor_persoana_urcare, 1 s
   "Scara2_DB_senzor_persoana_coborare" : Bool = PLC Scara2_DB.senzor_persoana_coborare, 1 s
   "Scara3_DB_senzor_persoana_urcare" : Bool = PLC Scara3_DB.senzor_persoana_urcare, 1 s
   "Scara3_DB_senzor_persoana_coborare" : Bool = PLC Scara3_DB.senzor_persoana_coborare, 1 s
   "Scara4_DB_senzor_persoana_urcare" : Bool = PLC Scara4_DB.senzor_persoana_urcare, 1 s
   "Scara4_DB_senzor_persoana_coborare" : Bool = PLC Scara4_DB.senzor_persoana_coborare, 1 s
   "HMI_timp_secunde_u_2" : Time = PLC HMI.timp_secunde_u_2, 1 s
   "HMI_timp_secunde_c_2" : Time = PLC HMI.timp_secunde_c_2, 1 s
   "HMI_timp_secunde_c_3" : Time = PLC HMI.timp_secunde_c_3, 1 s
   "HMI_timp_secunde_u_3" : Time = PLC HMI.timp_secunde_u_3, 1 s
   "HMI_timp_secunde_u_4" : Time = PLC HMI.timp_secunde_u_4, 1 s
   "HMI_timp_secunde_c_4" : Time = PLC HMI.timp_secunde_c_4, 1 s
   "Avarii_reset_avarie_2" : Bool = PLC Avarii.reset_avarie_2, 1 s

discrete alarms
   1: 'ESD', class Errors, trigger "Alarme_gather" bit 0
   2: 'Avarie la scara 1', class Errors, trigger "Alarme_gather" bit 1
   3: 'Avarie la scara 2', class Errors, trigger "Alarme_gather" bit 2
   4: 'Avarie la scara 3', class Errors, trigger "Alarme_gather" bit 3
   5: 'Avarie la scara 4', class Errors, trigger "Alarme_gather" bit 4

text list "Mod": 0 'Coborare'; 1 'Urcare'

screen "Main" 800x480, template "Template_1"
   TextField "Text field_1" at 73,18 size 58x22; Text 'Scari 1'
   Button "Button_1" at 41,57 size 31x28; TextOff 'ESD'
      Appearance <- "Avarii_btn_esd"
      on Press: SetBit("Avarii_btn_esd")
   Button "Button_2" at 41,84 size 31x28; TextOff 'Av.'
      Appearance <- "Avarii_btn_avarie_1"
      on Press: SetBit("Avarii_btn_avarie_1")
   Button "Button_3" at 71,57 size 31x28; TextOff 'Res'
      Appearance <- "Avarii_reset_esd"
      on Press: SetBit("Avarii_reset_esd")
   Button "Button_4" at 71,84 size 31x28; TextOff 'Res'
      Appearance <- "Avarii_reset_avarie_1"
      on Press: SetBit("Avarii_reset_avarie_1")
   Circle "Circle_1" at 10,58 size 25x25
      Appearance <- "Avarii_esd"
   Circle "Circle_2" at 10,86 size 25x25
      Appearance <- "Avarii_avarie_1"
   Rectangle "Rectangle_1" at 131,57 size 45x28
      Appearance <- "Scara1_DB_urcare_HMI"
   TextField "Text field_2" at 138,61 size 30x20; Text 'Urc.'
      Appearance <- "Scara1_DB_urcare_HMI"
   Rectangle "Rectangle_2" at 131,84 size 45x28
      Appearance <- "Scara1_DB_coborare_HMI"
   TextField "Text field_3" at 138,88 size 33x20; Text 'Cob.'
      Appearance <- "Scara1_DB_coborare_HMI"
   Button "Button_5" at 36,278 size 45x32; TextOff 'Start'
      Appearance <- "Scara1_DB_btn_start"
      on Press: SetBit("Scara1_DB_btn_start")
   SymbolicIOField "Symbolic I/O field_1" at 56,189 size 96x32; TextOff '0'; TextOn '1'; TextList "Mod"
      ProcessValue <- "Scara1_DB_mod"
      Visibility <- "Scara1_DB_btn_start"
   TextField "Text field_4" at 54,237 size 37x20; Text 'Mod:'
   Button "Button_6" at 36,309 size 45x32; TextOff 'Stop'
      Appearance <- "Scara1_DB_btn_stop"
      on Press: SetBit("Scara1_DB_btn_stop")
   Button "Button_7" at 19,379 size 72x32; TextOff 'Pers. urc.'
      on Press: SetBit("Scara1_DB_senzor_persoana_urcare")
      Appearance <- "Scara1_DB_senzor_persoana_urcare"
   Button "Button_8" at 19,408 size 72x32; TextOff 'Pers. cob.'
      Appearance <- "Scara1_DB_senzor_persoana_coborare"
      on Press: SetBit("Scara1_DB_senzor_persoana_coborare")
   TextField "Text field_5" at 102,357 size 93x20; Text 'Time elapsed:'
      Visibility <- "HMI_time_elapsed_HMI"
   IOField "I/O field_1" at 111,381 size 74x26; FormatPattern 9999; Unit s
      Visibility <- "Scara1_DB_senzor_persoana_urcare"
      ProcessValue <- "HMI_timp_secunde_u_1"
   IOField "I/O field_2" at 110,413 size 74x26; FormatPattern 9999; Unit s
      Visibility <- "Scara1_DB_senzor_persoana_coborare"
      ProcessValue <- "HMI_timp_secunde_c_1"
   Circle "Circle_3" at 116,290 size 48x48
      Appearance <- "HMI_pornit_HMI"
   TextField "Text field_6" at 118,269 size 44x20; Text 'Pornit'
   TextField "Text field_7" at 96,237 size 48x20; Text 'Urcare'
      Visibility <- "Scara1_DB_urcare_HMI"
   TextField "Text field_8" at 95,237 size 65x20; Text 'Coborare'
      Visibility <- "Scara1_DB_coborare_HMI"
   TextField "Text field_9" at 51,140 size 49x20; Text 'Motor:'
   Circle "Circle_4" at 116,128 size 48x48
      Appearance <- "HMI_mod_motor"
   TextField "Text field_10" at 275,18 size 58x22; Text 'Scari 2'
   Button "Button_9" at 243,57 size 31x28; TextOff 'ESD'
      on Press: SetBit("Avarii_btn_esd")
      Appearance <- "Avarii_btn_esd"
   Button "Button_10" at 243,84 size 31x28; TextOff 'Av.'
      on Press: SetBit("Avarii_btn_avarie_2")
      Appearance <- "Avarii_btn_avarie_2"
   Button "Button_11" at 273,57 size 31x28; TextOff 'Res'
      on Press: SetBit("Avarii_reset_esd")
      Appearance <- "Avarii_reset_esd"
   Button "Button_12" at 273,84 size 31x28; TextOff 'Res'
      on Press: SetBit("Avarii_reset_avarie_2")
      Appearance <- "Avarii_reset_avarie_2"
   Circle "Circle_5" at 212,58 size 25x25
      Appearance <- "Avarii_esd"
   Circle "Circle_6" at 212,86 size 25x25
      Appearance <- "Avarii_avarie_2"
   Rectangle "Rectangle_3" at 333,57 size 45x28
      Appearance <- "Scara2_DB_urcare_HMI"
   TextField "Text field_11" at 340,61 size 30x20; Text 'Urc.'
      Appearance <- "Scara2_DB_urcare_HMI"
   Rectangle "Rectangle_4" at 333,84 size 45x28
      Appearance <- "Scara2_DB_coborare_HMI"
   TextField "Text field_12" at 340,88 size 33x20; Text 'Cob.'
      Appearance <- "Scara2_DB_coborare_HMI"
   Button "Button_13" at 238,278 size 45x32; TextOff 'Start'
      on Press: SetBit("Scara2_DB_btn_start")
      Appearance <- "Scara2_DB_btn_start"
   SymbolicIOField "Symbolic I/O field_2" at 258,189 size 96x32; TextOn '1'; TextOff '0'; TextList "Mod"
      ProcessValue <- "Scara2_DB_mod"
      Visibility <- "Scara2_DB_btn_start"
   TextField "Text field_13" at 256,237 size 37x20; Text 'Mod:'
   Button "Button_14" at 238,309 size 45x32; TextOff 'Stop'
      on Press: SetBit("Scara2_DB_btn_stop")
      Appearance <- "Scara2_DB_btn_stop"
   Button "Button_15" at 221,379 size 72x32; TextOff 'Pers. urc.'
      on Press: SetBit("Scara2_DB_senzor_persoana_urcare")
      Appearance <- "Scara2_DB_senzor_persoana_urcare"
   Button "Button_16" at 221,408 size 72x32; TextOff 'Pers. cob.'
      on Press: SetBit("Scara2_DB_senzor_persoana_coborare")
      Appearance <- "Scara2_DB_senzor_persoana_coborare"
   TextField "Text field_14" at 304,357 size 93x20; Text 'Time elapsed:'
      Visibility <- "HMI_time_elapsed_HMI_2"
   IOField "I/O field_3" at 313,381 size 74x26; FormatPattern 9999; Unit s
      Visibility <- "Scara2_DB_senzor_persoana_urcare"
      ProcessValue <- "HMI_timp_secunde_u_2"
   IOField "I/O field_4" at 312,413 size 74x26; FormatPattern 9999; Unit s
      Visibility <- "Scara2_DB_senzor_persoana_coborare"
      ProcessValue <- "HMI_timp_secunde_c_2"
   Circle "Circle_7" at 318,290 size 48x48
      Appearance <- "HMI_pornit_HMI_2"
   TextField "Text field_15" at 320,269 size 44x20; Text 'Pornit'
   TextField "Text field_16" at 298,237 size 48x20; Text 'Urcare'
      Visibility <- "Scara2_DB_urcare_HMI"
   TextField "Text field_17" at 297,237 size 65x20; Text 'Coborare'
      Visibility <- "Scara2_DB_coborare_HMI"
   TextField "Text field_18" at 253,140 size 49x20; Text 'Motor:'
   Circle "Circle_8" at 318,128 size 48x48
      Appearance <- "HMI_mod_motor_2"
   TextField "Text field_19" at 474,18 size 58x22; Text 'Scari 3'
   Button "Button_17" at 442,57 size 31x28; TextOff 'ESD'
      on Press: SetBit("Avarii_btn_esd")
      Appearance <- "Avarii_btn_esd"
   Button "Button_18" at 442,84 size 31x28; TextOff 'Av.'
      on Press: SetBit("Avarii_btn_avarie_3")
      Appearance <- "Avarii_btn_avarie_3"
   Button "Button_19" at 472,57 size 31x28; TextOff 'Res'
      on Press: SetBit("Avarii_reset_esd")
      Appearance <- "Avarii_reset_esd"
   Button "Button_20" at 472,84 size 31x28; TextOff 'Res'
      on Press: SetBit("Avarii_reset_avarie_3")
      Appearance <- "Avarii_reset_avarie_3"
   Circle "Circle_9" at 411,58 size 25x25
      Appearance <- "Avarii_esd"
   Circle "Circle_10" at 411,86 size 25x25
      Appearance <- "Avarii_avarie_3"
   Rectangle "Rectangle_5" at 532,57 size 45x28
      Appearance <- "Scara3_DB_urcare_HMI"
   TextField "Text field_20" at 539,61 size 30x20; Text 'Urc.'
      Appearance <- "Scara3_DB_urcare_HMI"
   Rectangle "Rectangle_6" at 532,84 size 45x28
      Appearance <- "Scara3_DB_coborare_HMI"
   TextField "Text field_21" at 539,88 size 33x20; Text 'Cob.'
      Appearance <- "Scara3_DB_coborare_HMI"
   Button "Button_21" at 437,278 size 45x32; TextOff 'Start'
      on Press: SetBit("Scara3_DB_btn_start")
      Appearance <- "Scara3_DB_btn_start"
   SymbolicIOField "Symbolic I/O field_3" at 457,189 size 96x32; TextOn '1'; TextOff '0'; TextList "Mod"
      ProcessValue <- "Scara3_DB_mod"
      Visibility <- "Scara3_DB_btn_start"
   TextField "Text field_22" at 455,237 size 37x20; Text 'Mod:'
   Button "Button_22" at 437,309 size 45x32; TextOff 'Stop'
      on Press: SetBit("Scara3_DB_btn_stop")
      Appearance <- "Scara3_DB_btn_stop"
   Button "Button_23" at 420,379 size 72x32; TextOff 'Pers. urc.'
      on Press: SetBit("Scara3_DB_senzor_persoana_urcare")
      Appearance <- "Scara3_DB_senzor_persoana_urcare"
   Button "Button_24" at 420,408 size 72x32; TextOff 'Pers. cob.'
      on Press: SetBit("Scara3_DB_senzor_persoana_coborare")
      Appearance <- "Scara3_DB_senzor_persoana_coborare"
   TextField "Text field_23" at 503,357 size 93x20; Text 'Time elapsed:'
      Visibility <- "HMI_time_elapsed_HMI_3"
   IOField "I/O field_5" at 512,381 size 74x26; FormatPattern 9999; Unit s
      Visibility <- "Scara3_DB_senzor_persoana_urcare"
      ProcessValue <- "HMI_timp_secunde_u_3"
   IOField "I/O field_6" at 511,413 size 74x26; FormatPattern 9999; Unit s
      Visibility <- "Scara3_DB_senzor_persoana_coborare"
      ProcessValue <- "HMI_timp_secunde_c_3"
   Circle "Circle_11" at 517,290 size 48x48
      Appearance <- "HMI_pornit_HMI_3"
   TextField "Text field_24" at 519,269 size 44x20; Text 'Pornit'
   TextField "Text field_25" at 497,237 size 48x20; Text 'Urcare'
      Visibility <- "Scara3_DB_urcare_HMI"
   TextField "Text field_26" at 495,237 size 65x20; Text 'Coborare'
      Visibility <- "Scara3_DB_coborare_HMI"
   TextField "Text field_27" at 452,140 size 49x20; Text 'Motor:'
   Circle "Circle_12" at 517,128 size 48x48
      Appearance <- "HMI_mod_motor_3"
   TextField "Text field_28" at 674,18 size 58x22; Text 'Scari 4'
   Button "Button_25" at 642,57 size 31x28; TextOff 'ESD'
      on Press: SetBit("Avarii_btn_esd")
      Appearance <- "Avarii_btn_esd"
   Button "Button_26" at 642,84 size 31x28; TextOff 'Av.'
      on Press: SetBit("Avarii_btn_avarie_4")
      Appearance <- "Avarii_btn_avarie_4"
   Button "Button_27" at 672,57 size 31x28; TextOff 'Res'
      on Press: SetBit("Avarii_reset_esd")
      Appearance <- "Avarii_reset_esd"
   Button "Button_28" at 672,84 size 31x28; TextOff 'Res'
      on Press: SetBit("Avarii_reset_avarie_4")
      Appearance <- "Avarii_reset_avarie_4"
   Circle "Circle_13" at 611,58 size 25x25
      Appearance <- "Avarii_esd"
   Circle "Circle_14" at 611,86 size 25x25
      Appearance <- "Avarii_avarie_4"
   Rectangle "Rectangle_7" at 732,57 size 45x28
      Appearance <- "Scara4_DB_urcare_HMI"
   TextField "Text field_29" at 739,61 size 30x20; Text 'Urc.'
      Appearance <- "Scara4_DB_urcare_HMI"
   Rectangle "Rectangle_8" at 732,84 size 45x28
      Appearance <- "Scara4_DB_coborare_HMI"
   TextField "Text field_30" at 739,88 size 33x20; Text 'Cob.'
      Appearance <- "Scara4_DB_coborare_HMI"
   Button "Button_29" at 637,278 size 45x32; TextOff 'Start'
      on Press: SetBit("Scara4_DB_btn_start")
      Appearance <- "Scara4_DB_btn_start"
   SymbolicIOField "Symbolic I/O field_4" at 657,189 size 96x32; TextOn '1'; TextOff '0'; TextList "Mod"
      ProcessValue <- "Scara4_DB_mod"
      Visibility <- "Scara4_DB_btn_start"
   TextField "Text field_31" at 655,237 size 37x20; Text 'Mod:'
   Button "Button_30" at 637,309 size 45x32; TextOff 'Stop'
      on Press: SetBit("Scara4_DB_btn_stop")
      Appearance <- "Scara4_DB_btn_stop"
   Button "Button_31" at 620,379 size 72x32; TextOff 'Pers. urc.'
      on Press: SetBit("Scara4_DB_senzor_persoana_urcare")
      Appearance <- "Scara4_DB_senzor_persoana_urcare"
   Button "Button_32" at 620,408 size 72x32; TextOff 'Pers. cob.'
      on Press: SetBit("Scara4_DB_senzor_persoana_coborare")
      Appearance <- "Scara4_DB_senzor_persoana_coborare"
   TextField "Text field_32" at 703,357 size 93x20; Text 'Time elapsed:'
      Visibility <- "HMI_time_elapsed_HMI_4"
   IOField "I/O field_7" at 712,381 size 74x26; FormatPattern 9999; Unit s
      Visibility <- "Scara4_DB_senzor_persoana_urcare"
      ProcessValue <- "HMI_timp_secunde_u_4"
   IOField "I/O field_8" at 711,413 size 74x26; FormatPattern 9999; Unit s
      Visibility <- "Scara4_DB_senzor_persoana_coborare"
      ProcessValue <- "HMI_timp_secunde_c_4"
   Circle "Circle_15" at 717,290 size 48x48
      Appearance <- "HMI_pornit_HMI_4"
   TextField "Text field_33" at 719,269 size 44x20; Text 'Pornit'
   TextField "Text field_34" at 697,237 size 48x20; Text 'Urcare'
      Visibility <- "Scara4_DB_urcare_HMI"
   TextField "Text field_35" at 696,237 size 65x20; Text 'Coborare'
      Visibility <- "Scara4_DB_coborare_HMI"
   TextField "Text field_36" at 652,140 size 49x20; Text 'Motor:'
   Circle "Circle_16" at 717,128 size 48x48
      Appearance <- "HMI_mod_motor_4"
*)

(* ===== HMI "HMI_RT_2" =====
system functions are stored by id; their names below are inferred from use
connection "HMI_Connection_2": ETHERNET, SMART_S7_1500_OMS

HMI tags "Default tag table"
   "Alarme_gather" : Word = PLC Alarme.gather, 1 s
   "Usa_Metrou1_DB_deschide_2" : Bool = PLC Usa_Metrou1_DB.deschide_2, 1 s
   "Usa_Metrou1_DB_senzor_laser_1" : Bool = PLC Usa_Metrou1_DB.senzor_laser_1, 1 s
   "Usa_Metrou1_DB_senzor_laser_2" : Bool = PLC Usa_Metrou1_DB.senzor_laser_2, 1 s
   "Usa_Metrou1_DB_deschide_1" : Bool = PLC Usa_Metrou1_DB.deschide_1, 1 s
   "Usa_Metrou1_DB_sunet_buzzer" : Bool = PLC Usa_Metrou1_DB.sunet_buzzer, 1 s
   "Usa_Metrou1_DB_confirmare_primita" : Bool = PLC Usa_Metrou1_DB.confirmare_primita, 1 s
   "Usa_Metrou1_DB_trimite_confirmare" : Bool = PLC Usa_Metrou1_DB.trimite_confirmare, 1 s
   "Avarii_esd" : Bool = PLC Avarii.esd, 1 s
   "Avarii_btn_esd" : Bool = PLC Avarii.btn_esd, 1 s
   "Avarii_reset_esd" : Bool = PLC Avarii.reset_esd, 1 s
   "Avarii_reset_avaie_usa_1" : Bool = PLC Avarii.reset_avaie_usa_1, 1 s
   "Avarii_btn_avarie_usa_1" : Bool = PLC Avarii.btn_avarie_usa_1, 1 s
   "Avarii_avarie_usa_1" : Bool = PLC Avarii.avarie_usa_1, 1 s
   "Usa_Metrou1_DB_secventa_pornita" : Bool = PLC Usa_Metrou1_DB.secventa_pornita, 1 s
   "Usa_Metrou1_DB_mod" : DInt = PLC Usa_Metrou1_DB.mod, 1 s
   "Usa_Metrou1_DB_usi_inchise" : Bool = PLC Usa_Metrou1_DB.usi_inchise, 1 s
   "Usa_Metrou1_DB_vizibilitate_mod_02" : Bool = PLC Usa_Metrou1_DB.vizibilitate_mod_02, 1 s

discrete alarms
   1: 'ESD', class Errors, trigger "Alarme_gather" bit 0
   2: 'Avarie usa 1', class Errors, trigger "Alarme_gather" bit 1
   3: 'Avarie usa 2', class Errors, trigger "Alarme_gather" bit 2
   4: 'Avarie usa 3', class Errors, trigger "Alarme_gather" bit 3

text list "Mod": 0 'Spre metrou'; 1 'Spre iesire'; 2 'Mixt'

screen "Usa1" 800x480, template "Template_1"
   Button "Button_1" at 238,328 size 54x32; TextOff 'Laser 1'
      on Press: SetBit("Usa_Metrou1_DB_senzor_laser_1")
      on Release: ResetBit("Usa_Metrou1_DB_senzor_laser_1")
      Appearance <- "Usa_Metrou1_DB_senzor_laser_1"
   Button "Button_2" at 238,134 size 54x32; TextOff 'Laser 2'
      on Release: ResetBit("Usa_Metrou1_DB_senzor_laser_2")
      on Press: SetBit("Usa_Metrou1_DB_senzor_laser_2")
      Appearance <- "Usa_Metrou1_DB_senzor_laser_2"
   Rectangle "Rectangle_1" at 541,139 size 28x28
      Appearance <- "Usa_Metrou1_DB_sunet_buzzer"
      Visibility <- "Usa_Metrou1_DB_vizibilitate_mod_02"
   Button "Button_3" at 502,325 size 45x32; TextOff 'Plata'
      on Press: SetBit("Usa_Metrou1_DB_trimite_confirmare")
      Visibility <- "Usa_Metrou1_DB_vizibilitate_mod_02"
      Appearance <- "Usa_Metrou1_DB_trimite_confirmare"
   TextField "Text field_2" at 24,76 size 43x20; Text 'Peron'
   TextField "Text field_3" at 373,76 size 43x20; Text 'Peron'
   TextField "Text field_4" at 728,76 size 43x20; Text 'Peron'
   TextField "Text field_5" at 99,441 size 37x20; Text 'Scari'
   TextField "Text field_6" at 659,441 size 37x20; Text 'Scari'
   SymbolicIOField "Symbolic I/O field_1" at 332,392 size 123x32; TextOff '0'; TextOn '1'; TextList "Mod"
      Visibility <- "Usa_Metrou1_DB_secventa_pornita"
      ProcessValue <- "Usa_Metrou1_DB_mod"
   TextField "Text field_7" at 376,367 size 32x20; Text 'Mod'
      Visibility <- "Usa_Metrou1_DB_secventa_pornita"
   TextField "Text field_8" at 360,102 size 70x32; Text 'Usa 1'
   Rectangle "Rectangle_37" at 300,236 size 85x20
      Visibility <- "Usa_Metrou1_DB_usi_inchise"
   Rectangle "Rectangle_38" at 405,236 size 85x20
      Visibility <- "Usa_Metrou1_DB_usi_inchise"
   Rectangle "Rectangle_39" at 300,164 size 21x73
      Visibility <- "Usa_Metrou1_DB_deschide_1"
   Rectangle "Rectangle_40" at 469,164 size 21x73
      Visibility <- "Usa_Metrou1_DB_deschide_1"
   Rectangle "Rectangle_41" at 300,255 size 21x73
      Visibility <- "Usa_Metrou1_DB_deschide_2"
   Rectangle "Rectangle_42" at 469,255 size 21x73
      Visibility <- "Usa_Metrou1_DB_deschide_2"
   Button "Button_4" at 51,134 size 31x28; TextOff 'ESD'
      on Press: SetBit("Avarii_btn_esd")
      Appearance <- "Avarii_btn_esd"
   Button "Button_5" at 51,161 size 31x28; TextOff 'Av.'
      on Press: SetBit("Avarii_btn_avarie_usa_1")
      Appearance <- "Avarii_btn_avarie_usa_1"
   Button "Button_6" at 81,134 size 31x28; TextOff 'Res'
      on Press: SetBit("Avarii_reset_esd")
      Appearance <- "Avarii_reset_esd"
      on Release: ResetBit("Avarii_reset_esd")
   Button "Button_7" at 81,161 size 31x28; TextOff 'Res'
      on Press: SetBit("Avarii_reset_avaie_usa_1")
      on Release: ResetBit("Avarii_reset_avaie_usa_1")
      Appearance <- "Avarii_reset_avaie_usa_1"
   Circle "Circle_1" at 20,135 size 25x25
      Appearance <- "Avarii_esd"
   Circle "Circle_3" at 20,163 size 25x25
      Appearance <- "Avarii_avarie_usa_1"
   TextField "Text field_1" at 530,114 size 49x20; Text 'Buzzer'
      Visibility <- "Usa_Metrou1_DB_vizibilitate_mod_02"
*)